LIN {X 0,Y 165.279,Z 285.697,A -85,B 0,C 180,E1 -23392.213,E2 -23392.213} C_VEL
LIN {X 0,Y 165.239,Z 285.426,A -85,B 0,C 180,E1 -23392.672,E2 -23392.672} C_VEL
LIN {X 0,Y 165.636,Z 284.894,A -85,B 0,C 180,E1 -23400.003,E2 -23400.003} C_VEL
LIN {X 0,Y 165.274,Z 285.304,A -85,B 0,C 180,E1 -23407.332,E2 -23407.332} C_VEL
LIN {X 0,Y 165.239,Z 285.88,A -85,B 0,C 180,E1 -23411.981,E2 -23411.981} C_VEL
LIN {X 0,Y 165.204,Z 286.851,A -85,B 0,C 180,E1 -23417.328,E2 -23417.328} C_VEL
LIN {X 0,Y 165.354,Z 287.875,A -85,B 0,C 180,E1 -23420.922,E2 -23420.922} C_VEL
LIN {X 0,Y 166.724,Z 291.129,A -85,B 0,C 180,E1 -23423.281,E2 -23423.281} C_VEL
LIN {X 0,Y 169.93,Z 294.587,A -85,B 0,C 180,E1 -23427.064,E2 -23427.064} C_VEL
LIN {X 0,Y 171.948,Z 298.713,A -85,B 0,C 180,E1 -23429.543,E2 -23429.543} C_VEL
LIN {X 0,Y 174.222,Z 301.462,A -85,B 0,C 180,E1 -23431.708,E2 -23431.708} C_VEL
LIN {X 0,Y 176.103,Z 305.449,A -85,B 0,C 180,E1 -23433.736,E2 -23433.736} C_VEL
LIN {X 0,Y 177.62,Z 307.849,A -85,B 0,C 180,E1 -23435.139,E2 -23435.139} C_VEL
LIN {X 0,Y 180.387,Z 313.585,A -85,B 0,C 180,E1 -23437.856,E2 -23437.856} C_VEL
LIN {X 0,Y 183.198,Z 320.279,A -85,B 0,C 180,E1 -23440.708,E2 -23440.708} C_VEL
LIN {X 0,Y 185.902,Z 327.653,A -85,B 0,C 180,E1 -23443.628,E2 -23443.628} C_VEL
LIN {X 0,Y 187.357,Z 334.16,A -85,B 0,C 180,E1 -23445.893,E2 -23445.893} C_VEL
LIN {X 0,Y 187.851,Z 342.319,A -85,B 0,C 180,E1 -23448.442,E2 -23448.442} C_VEL
LIN {X 0,Y 187.472,Z 350.553,A -85,B 0,C 180,E1 -23451.036,E2 -23451.036} C_VEL
LIN {X 0,Y 186.501,Z 358.181,A -85,B 0,C 180,E1 -23453.594,E2 -23453.594} C_VEL
LIN {X 0,Y 185.205,Z 363.138,A -85,B 0,C 180,E1 -23455.306,E2 -23455.306} C_VEL
LIN {X 0,Y 180.202,Z 371.77,A -85,B 0,C 180,E1 -23458.231,E2 -23458.231} C_VEL
LIN {X 0,Y 175.803,Z 378.681,A -85,B 0,C 180,E1 -23461.334,E2 -23461.334} C_VEL
LIN {X 0,Y 172.088,Z 384.243,A -85,B 0,C 180,E1 -23464.608,E2 -23464.608} C_VEL
LIN {X 0,Y 168.804,Z 388.644,A -85,B 0,C 180,E1 -23467.994,E2 -23467.994} C_VEL
LIN {X 0,Y 166.897,Z 390.981,A -85,B 0,C 180,E1 -23470.314,E2 -23470.314} C_VEL
LIN {X 0,Y 165.302,Z 392.899,A -85,B 0,C 180,E1 -23472.686,E2 -23472.686} C_VEL
LIN {X 0,Y 164.118,Z 394.399,A -85,B 0,C 180,E1 -23475.112,E2 -23475.112} C_VEL
LIN {X 0,Y 162.46,Z 396.157,A -85,B 0,C 180,E1 -23480.036,E2 -23480.036} C_VEL
LIN {X 0,Y 161.856,Z 396.404,A -85,B 0,C 180,E1 -23485.018,E2 -23485.018} C_VEL
LIN {X 0,Y 161.843,Z 395.911,A -85,B 0,C 180,E1 -23487.511,E2 -23487.511} C_VEL
LIN {X 0,Y 161.942,Z 395.021,A -85,B 0,C 180,E1 -23490,E2 -23490} C_VEL
LIN {X 0,Y 161.84,Z 393.556,A -85,B 0,C 180,E1 -23492.769,E2 -23492.769} C_VEL
LIN {X 0,Y 161.976,Z 390.939,A -85,B 0,C 180,E1 -23496.227,E2 -23496.227} C_VEL
LIN {X 0,Y 162.403,Z 387.105,A -85,B 0,C 180,E1 -23499.968,E2 -23499.968} C_VEL
LIN {X 0,Y 163.312,Z 382.12,A -85,B 0,C 180,E1 -23503.691,E2 -23503.691} C_VEL
LIN {X 0,Y 164.882,Z 375.841,A -85,B 0,C 180,E1 -23507.359,E2 -23507.359} C_VEL
LIN {X 0,Y 167.078,Z 367.691,A -85,B 0,C 180,E1 -23511.067,E2 -23511.067} C_VEL
LIN {X 0,Y 168.85,Z 360.58,A -85,B 0,C 180,E1 -23513.689,E2 -23513.689} C_VEL
LIN {X 0,Y 171.428,Z 351.112,A -85,B 0,C 180,E1 -23516.477,E2 -23516.477} C_VEL
LIN {X 0,Y 172.232,Z 346.562,A -85,B 0,C 180,E1 -23517.655,E2 -23517.655} C_VEL
LIN {X 0,Y 172.3,Z 345.493,A -85,B 0,C 180,E1 -23517.932,E2 -23517.932} C_VEL
LIN {X 0,Y 171.915,Z 340.91,A -85,B 0,C 180,E1 -23519.161,E2 -23519.161} C_VEL
LIN {X 0,Y 170.545,Z 336.486,A -85,B 0,C 180,E1 -23520.408,E2 -23520.408} C_VEL
LIN {X 0,Y 166.885,Z 327.585,A -85,B 0,C 180,E1 -23522.844,E2 -23522.844} C_VEL
LIN {X 0,Y 165.579,Z 322.739,A -85,B 0,C 180,E1 -23523.969,E2 -23523.969} C_VEL
LIN {X 0,Y 165.325,Z 321.027,A -85,B 0,C 180,E1 -23524.313,E2 -23524.313} C_VEL
LIN {X 0,Y 163.739,Z 309.046,A -85,B 0,C 180,E1 -23526.448,E2 -23526.448} C_VEL
LIN {X 0,Y 161.215,Z 297.421,A -85,B 0,C 180,E1 -23528.304,E2 -23528.304} C_VEL
LIN {X 0,Y 159.652,Z 293.515,A -85,B 0,C 180,E1 -23528.995,E2 -23528.995} C_VEL
LIN {X 0,Y 158.483,Z 290.377,A -85,B 0,C 180,E1 -23529.519,E2 -23529.519} C_VEL
LIN {X 0,Y 158.438,Z 289.902,A -85,B 0,C 180,E1 -23529.716,E2 -23529.716} C_VEL
LIN {X 0,Y 157.715,Z 286.321,A -85,B 0,C 180,E1 -23535.477,E2 -23535.477} C_VEL
LIN {X 0,Y 157.262,Z 283.904,A -85,B 0,C 180,E1 -23539.885,E2 -23539.885} C_VEL
LIN {X 0,Y 157.276,Z 283.897,A -85,B 0,C 180,E1 -23544.482,E2 -23544.482} C_VEL
LIN {X 0,Y 157.284,Z 283.893,A -85,B 0,C 180,E1 -23548.1,E2 -23548.1} C_VEL
LIN {X 0,Y 157.31,Z 283.89,A -85,B 0,C 180,E1 -23553.461,E2 -23553.461} C_VEL
LIN {X 0,Y 157.392,Z 283.881,A -85,B 0,C 180,E1 -23559.667,E2 -23559.667} C_VEL
LIN {X 0,Y 157.44,Z 283.875,A -85,B 0,C 180,E1 -23564.461,E2 -23564.461} C_VEL
LIN {X 0,Y 157.688,Z 283.837,A -85,B 0,C 180,E1 -23569.728,E2 -23569.728} C_VEL
LIN {X 0,Y 157.765,Z 283.836,A -85,B 0,C 180,E1 -23572.317,E2 -23572.317} C_VEL
LIN {X 0,Y 158.255,Z 283.735,A -85,B 0,C 180,E1 -23579.997,E2 -23579.997} C_VEL
LIN {X 0,Y 157.806,Z 283.826,A -85,B 0,C 180,E1 -23587.675,E2 -23587.675} C_VEL
LIN {X 0,Y 157.668,Z 283.84,A -85,B 0,C 180,E1 -23591.298,E2 -23591.298} C_VEL
LIN {X 0,Y 157.448,Z 283.866,A -85,B 0,C 180,E1 -23595.531,E2 -23595.531} C_VEL
LIN {X 0,Y 157.364,Z 283.883,A -85,B 0,C 180,E1 -23600.93,E2 -23600.93} C_VEL
LIN {X 0,Y 157.305,Z 283.888,A -85,B 0,C 180,E1 -23606.679,E2 -23606.679} C_VEL
LIN {X 0,Y 157.271,Z 283.89,A -85,B 0,C 180,E1 -23612.424,E2 -23612.424} C_VEL
LIN {X 0,Y 157.318,Z 283.878,A -85,B 0,C 180,E1 -23616.475,E2 -23616.475} C_VEL
LIN {X 0,Y 157.264,Z 283.887,A -85,B 0,C 180,E1 -23622.089,E2 -23622.089} C_VEL
LIN {X 0,Y 157.223,Z 283.892,A -85,B 0,C 180,E1 -23627.894,E2 -23627.894} C_VEL
LIN {X 0,Y 157.272,Z 283.891,A -85,B 0,C 180,E1 -23633.543,E2 -23633.543} C_VEL
LIN {X 0,Y 157.276,Z 283.894,A -85,B 0,C 180,E1 -23638.1,E2 -23638.1} C_VEL
LIN {X 0,Y 157.298,Z 283.954,A -85,B 0,C 180,E1 -23643.32,E2 -23643.32} C_VEL
LIN {X 0,Y 158.336,Z 286.745,A -85,B 0,C 180,E1 -23643.813,E2 -23643.813} C_VEL
LIN {X 0,Y 159.794,Z 289.096,A -85,B 0,C 180,E1 -23644.361,E2 -23644.361} C_VEL
LIN {X 0,Y 161.784,Z 294.226,A -85,B 0,C 180,E1 -23645.342,E2 -23645.342} C_VEL
LIN {X 0,Y 164.927,Z 305.378,A -85,B 0,C 180,E1 -23647.449,E2 -23647.449} C_VEL
LIN {X 0,Y 166.797,Z 315.823,A -85,B 0,C 180,E1 -23649.548,E2 -23649.548} C_VEL
LIN {X 0,Y 167.906,Z 326.811,A -85,B 0,C 180,E1 -23652.02,E2 -23652.02} C_VEL
LIN {X 0,Y 167.891,Z 333.244,A -85,B 0,C 180,E1 -23653.587,E2 -23653.587} C_VEL
LIN {X 0,Y 165.068,Z 343.638,A -85,B 0,C 180,E1 -23656.144,E2 -23656.144} C_VEL
LIN {X 0,Y 162.84,Z 352.088,A -85,B 0,C 180,E1 -23658.801,E2 -23658.801} C_VEL
LIN {X 0,Y 160.566,Z 359.905,A -85,B 0,C 180,E1 -23661.822,E2 -23661.822} C_VEL
LIN {X 0,Y 158.265,Z 367.551,A -85,B 0,C 180,E1 -23665.543,E2 -23665.543} C_VEL
LIN {X 0,Y 156.935,Z 372.774,A -85,B 0,C 180,E1 -23668.717,E2 -23668.717} C_VEL
LIN {X 0,Y 155.776,Z 377.838,A -85,B 0,C 180,E1 -23672.586,E2 -23672.586} C_VEL
LIN {X 0,Y 154.956,Z 381.781,A -85,B 0,C 180,E1 -23676.51,E2 -23676.51} C_VEL
LIN {X 0,Y 154.432,Z 384.696,A -85,B 0,C 180,E1 -23680.488,E2 -23680.488} C_VEL
LIN {X 0,Y 154.39,Z 386.074,A -85,B 0,C 180,E1 -23683.156,E2 -23683.156} C_VEL
LIN {X 0,Y 154.746,Z 387.44,A -85,B 0,C 180,E1 -23687.507,E2 -23687.507} C_VEL
LIN {X 0,Y 155.396,Z 387.75,A -85,B 0,C 180,E1 -23691.211,E2 -23691.211} C_VEL
LIN {X 0,Y 156.252,Z 387.467,A -85,B 0,C 180,E1 -23693.878,E2 -23693.878} C_VEL
LIN {X 0,Y 157.494,Z 386.688,A -85,B 0,C 180,E1 -23696.822,E2 -23696.822} C_VEL
LIN {X 0,Y 160.357,Z 384.065,A -85,B 0,C 180,E1 -23701.73,E2 -23701.73} C_VEL
LIN {X 0,Y 162.836,Z 381.433,A -85,B 0,C 180,E1 -23704.917,E2 -23704.917} C_VEL
LIN {X 0,Y 167.024,Z 376.456,A -85,B 0,C 180,E1 -23709.135,E2 -23709.135} C_VEL
LIN {X 0,Y 171.629,Z 370.382,A -85,B 0,C 180,E1 -23712.834,E2 -23712.834} C_VEL
LIN {X 0,Y 176.146,Z 363.694,A -85,B 0,C 180,E1 -23715.903,E2 -23715.903} C_VEL
LIN {X 0,Y 181.013,Z 355.688,A -85,B 0,C 180,E1 -23718.701,E2 -23718.701} C_VEL
LIN {X 0,Y 182.586,Z 352.612,A -85,B 0,C 180,E1 -23719.661,E2 -23719.661} C_VEL
LIN {X 0,Y 183.295,Z 344.321,A -85,B 0,C 180,E1 -23722.89,E2 -23722.89} C_VEL
LIN {X 0,Y 183.118,Z 337.344,A -85,B 0,C 180,E1 -23725.525,E2 -23725.525} C_VEL
LIN {X 0,Y 182.209,Z 330.915,A -85,B 0,C 180,E1 -23728.053,E2 -23728.053} C_VEL
LIN {X 0,Y 180.3,Z 324.284,A -85,B 0,C 180,E1 -23730.936,E2 -23730.936} C_VEL
LIN {X 0,Y 177.754,Z 317.303,A -85,B 0,C 180,E1 -23734.223,E2 -23734.223} C_VEL
LIN {X 0,Y 175.156,Z 311.906,A -85,B 0,C 180,E1 -23737.163,E2 -23737.163} C_VEL
LIN {X 0,Y 172.885,Z 307.483,A -85,B 0,C 180,E1 -23739.789,E2 -23739.789} C_VEL
LIN {X 0,Y 170,Z 302.603,A -85,B 0,C 180,E1 -23743.182,E2 -23743.182} C_VEL
LIN {X 0,Y 167.954,Z 299.607,A -85,B 0,C 180,E1 -23745.694,E2 -23745.694} C_VEL
LIN {X 0,Y 167.153,Z 297.848,A -85,B 0,C 180,E1 -23746.942,E2 -23746.942} C_VEL
LIN {X 0,Y 164.506,Z 294.958,A -85,B 0,C 180,E1 -23750.629,E2 -23750.629} C_VEL
LIN {X 0,Y 163.297,Z 292.219,A -85,B 0,C 180,E1 -23753.206,E2 -23753.206} C_VEL
LIN {X 0,Y 160.482,Z 289.774,A -85,B 0,C 180,E1 -23760.003,E2 -23760.003} C_VEL
LIN {X 0,Y 159.59,Z 289.477,A -85,B 0,C 180,E1 -23765.056,E2 -23765.056} C_VEL
LIN {X 0,Y 159.736,Z 289.995,A -85,B 0,C 180,E1 -23769.5,E2 -23769.5} C_VEL
LIN {X 0,Y 163.477,Z 294.396,A -85,B 0,C 180,E1 -23780.119,E2 -23780.119} C_VEL
LIN {X 0,Y 164.634,Z 297.606,A -85,B 0,C 180,E1 -23782.597,E2 -23782.597} C_VEL
LIN {X 0,Y 167.62,Z 301.396,A -85,B 0,C 180,E1 -23786.625,E2 -23786.625} C_VEL
LIN {X 0,Y 168.954,Z 304.57,A -85,B 0,C 180,E1 -23788.583,E2 -23788.583} C_VEL
LIN {X 0,Y 171.064,Z 307.424,A -85,B 0,C 180,E1 -23790.904,E2 -23790.904} C_VEL
LIN {X 0,Y 172.593,Z 311.035,A -85,B 0,C 180,E1 -23792.85,E2 -23792.85} C_VEL
LIN {X 0,Y 174.036,Z 313.646,A -85,B 0,C 180,E1 -23794.43,E2 -23794.43} C_VEL
LIN {X 0,Y 177.073,Z 320.756,A -85,B 0,C 180,E1 -23797.967,E2 -23797.967} C_VEL
LIN {X 0,Y 179.999,Z 328.949,A -85,B 0,C 180,E1 -23801.59,E2 -23801.59} C_VEL
LIN {X 0,Y 181.606,Z 335.39,A -85,B 0,C 180,E1 -23804.157,E2 -23804.157} C_VEL
LIN {X 0,Y 182.117,Z 340.664,A -85,B 0,C 180,E1 -23806.004,E2 -23806.004} C_VEL
LIN {X 0,Y 181.912,Z 348.306,A -85,B 0,C 180,E1 -23808.539,E2 -23808.539} C_VEL
LIN {X 0,Y 180.859,Z 356.997,A -85,B 0,C 180,E1 -23811.558,E2 -23811.558} C_VEL
LIN {X 0,Y 179.336,Z 363.575,A -85,B 0,C 180,E1 -23813.998,E2 -23813.998} C_VEL
LIN {X 0,Y 174.219,Z 372.049,A -85,B 0,C 180,E1 -23817.004,E2 -23817.004} C_VEL
LIN {X 0,Y 169.599,Z 378.868,A -85,B 0,C 180,E1 -23820.182,E2 -23820.182} C_VEL
LIN {X 0,Y 165.702,Z 384.352,A -85,B 0,C 180,E1 -23823.556,E2 -23823.556} C_VEL
LIN {X 0,Y 162.216,Z 388.682,A -85,B 0,C 180,E1 -23827.051,E2 -23827.051} C_VEL
LIN {X 0,Y 160.216,Z 390.985,A -85,B 0,C 180,E1 -23829.457,E2 -23829.457} C_VEL
LIN {X 0,Y 158.515,Z 392.869,A -85,B 0,C 180,E1 -23831.92,E2 -23831.92} C_VEL
LIN {X 0,Y 156.214,Z 395.344,A -85,B 0,C 180,E1 -23837.001,E2 -23837.001} C_VEL
LIN {X 0,Y 154.98,Z 396.286,A -85,B 0,C 180,E1 -23842.181,E2 -23842.181} C_VEL
LIN {X 0,Y 154.765,Z 396.165,A -85,B 0,C 180,E1 -23844.789,E2 -23844.789} C_VEL
LIN {X 0,Y 154.749,Z 395.547,A -85,B 0,C 180,E1 -23847.69,E2 -23847.69} C_VEL
LIN {X 0,Y 154.86,Z 394.714,A -85,B 0,C 180,E1 -23850,E2 -23850} C_VEL
LIN {X 0,Y 154.747,Z 393.38,A -85,B 0,C 180,E1 -23852.603,E2 -23852.603} C_VEL
LIN {X 0,Y 154.902,Z 390.534,A -85,B 0,C 180,E1 -23856.513,E2 -23856.513} C_VEL
LIN {X 0,Y 155.4,Z 386.632,A -85,B 0,C 180,E1 -23860.422,E2 -23860.422} C_VEL
LIN {X 0,Y 156.383,Z 381.571,A -85,B 0,C 180,E1 -23864.31,E2 -23864.31} C_VEL
LIN {X 0,Y 158.055,Z 375.197,A -85,B 0,C 180,E1 -23868.135,E2 -23868.135} C_VEL
LIN {X 0,Y 160.353,Z 367.189,A -85,B 0,C 180,E1 -23871.872,E2 -23871.872} C_VEL
LIN {X 0,Y 161.778,Z 361.497,A -85,B 0,C 180,E1 -23874.085,E2 -23874.085} C_VEL
LIN {X 0,Y 164.457,Z 352.241,A -85,B 0,C 180,E1 -23877.003,E2 -23877.003} C_VEL
LIN {X 0,Y 165.445,Z 347.846,A -85,B 0,C 180,E1 -23878.201,E2 -23878.201} C_VEL
LIN {X 0,Y 165.907,Z 337.311,A -85,B 0,C 180,E1 -23880.89,E2 -23880.89} C_VEL
LIN {X 0,Y 165.735,Z 326.673,A -85,B 0,C 180,E1 -23883.205,E2 -23883.205} C_VEL
LIN {X 0,Y 165.325,Z 321.027,A -85,B 0,C 180,E1 -23884.313,E2 -23884.313} C_VEL
LIN {X 0,Y 164.169,Z 316.085,A -85,B 0,C 180,E1 -23885.362,E2 -23885.362} C_VEL
LIN {X 0,Y 162.1,Z 311.515,A -85,B 0,C 180,E1 -23886.482,E2 -23886.482} C_VEL
LIN {X 0,Y 155.231,Z 299.656,A -85,B 0,C 180,E1 -23889.493,E2 -23889.493} C_VEL
LIN {X 0,Y 153.815,Z 296.375,A -85,B 0,C 180,E1 -23890.169,E2 -23890.169} C_VEL
LIN {X 0,Y 152.408,Z 293.22,A -85,B 0,C 180,E1 -23890.811,E2 -23890.811} C_VEL
LIN {X 0,Y 151.237,Z 290.151,A -85,B 0,C 180,E1 -23891.381,E2 -23891.381} C_VEL
LIN {X 0,Y 151.175,Z 289.718,A -85,B 0,C 180,E1 -23891.501,E2 -23891.501} C_VEL
LIN {X 0,Y 150.68,Z 287.319,A -85,B 0,C 180,E1 -23895.599,E2 -23895.599} C_VEL
LIN {X 0,Y 150.217,Z 284.782,A -85,B 0,C 180,E1 -23900.394,E2 -23900.394} C_VEL
LIN {X 0,Y 150.187,Z 284.777,A -85,B 0,C 180,E1 -23905.834,E2 -23905.834} C_VEL
LIN {X 0,Y 150.192,Z 284.773,A -85,B 0,C 180,E1 -23909.017,E2 -23909.017} C_VEL
LIN {X 0,Y 150.24,Z 284.772,A -85,B 0,C 180,E1 -23912.72,E2 -23912.72} C_VEL
LIN {X 0,Y 150.35,Z 284.758,A -85,B 0,C 180,E1 -23919.207,E2 -23919.207} C_VEL
LIN {X 0,Y 150.351,Z 284.754,A -85,B 0,C 180,E1 -23923.709,E2 -23923.709} C_VEL
LIN {X 0,Y 150.61,Z 284.717,A -85,B 0,C 180,E1 -23929.239,E2 -23929.239} C_VEL
LIN {X 0,Y 150.702,Z 284.715,A -85,B 0,C 180,E1 -23931.955,E2 -23931.955} C_VEL
LIN {X 0,Y 151.215,Z 284.61,A -85,B 0,C 180,E1 -23939.997,E2 -23939.997} C_VEL
LIN {X 0,Y 150.74,Z 284.704,A -85,B 0,C 180,E1 -23948.037,E2 -23948.037} C_VEL
LIN {X 0,Y 150.602,Z 284.721,A -85,B 0,C 180,E1 -23951.488,E2 -23951.488} C_VEL
LIN {X 0,Y 150.355,Z 284.747,A -85,B 0,C 180,E1 -23956.284,E2 -23956.284} C_VEL
LIN {X 0,Y 150.345,Z 284.757,A -85,B 0,C 180,E1 -23960.789,E2 -23960.789} C_VEL
LIN {X 0,Y 150.236,Z 284.77,A -85,B 0,C 180,E1 -23967.278,E2 -23967.278} C_VEL
LIN {X 0,Y 150.212,Z 284.77,A -85,B 0,C 180,E1 -23972.632,E2 -23972.632} C_VEL
LIN {X 0,Y 150.228,Z 284.763,A -85,B 0,C 180,E1 -23977.453,E2 -23977.453} C_VEL
LIN {X 0,Y 150.209,Z 284.767,A -85,B 0,C 180,E1 -23981.531,E2 -23981.531} C_VEL
LIN {X 0,Y 150.16,Z 284.779,A -85,B 0,C 180,E1 -23985.409,E2 -23985.409} C_VEL
LIN {X 0,Y 150.158,Z 284.776,A -85,B 0,C 180,E1 -23989.062,E2 -23989.062} C_VEL
LIN {X 0,Y 150.207,Z 284.769,A -85,B 0,C 180,E1 -23992.688,E2 -23992.688} C_VEL
LIN {X 0,Y 150.202,Z 284.776,A -85,B 0,C 180,E1 -23997.369,E2 -23997.369} C_VEL
LIN {X 0,Y 150.218,Z 284.931,A -85,B 0,C 180,E1 -24001.537,E2 -24001.537} C_VEL
LIN {X 0,Y 151.328,Z 287.771,A -85,B 0,C 180,E1 -24002.102,E2 -24002.102} C_VEL
LIN {X 0,Y 152.91,Z 290.388,A -85,B 0,C 180,E1 -24002.777,E2 -24002.777} C_VEL
LIN {X 0,Y 155.092,Z 294.395,A -85,B 0,C 180,E1 -24003.773,E2 -24003.773} C_VEL
LIN {X 0,Y 158.216,Z 305.436,A -85,B 0,C 180,E1 -24006.011,E2 -24006.011} C_VEL
LIN {X 0,Y 160.146,Z 315.532,A -85,B 0,C 180,E1 -24008.179,E2 -24008.179} C_VEL
LIN {X 0,Y 161.307,Z 327.158,A -85,B 0,C 180,E1 -24010.928,E2 -24010.928} C_VEL
LIN {X 0,Y 161.399,Z 333.533,A -85,B 0,C 180,E1 -24012.581,E2 -24012.581} C_VEL
LIN {X 0,Y 158.469,Z 343.908,A -85,B 0,C 180,E1 -24015.226,E2 -24015.226} C_VEL
LIN {X 0,Y 155.866,Z 353.18,A -85,B 0,C 180,E1 -24018.293,E2 -24018.293} C_VEL
LIN {X 0,Y 153.119,Z 362.192,A -85,B 0,C 180,E1 -24022.085,E2 -24022.085} C_VEL
LIN {X 0,Y 150.827,Z 369.472,A -85,B 0,C 180,E1 -24025.992,E2 -24025.992} C_VEL
LIN {X 0,Y 149.296,Z 375.275,A -85,B 0,C 180,E1 -24030,E2 -24030} C_VEL
LIN {X 0,Y 148.244,Z 380.142,A -85,B 0,C 180,E1 -24034.395,E2 -24034.395} C_VEL
LIN {X 0,Y 147.562,Z 383.35,A -85,B 0,C 180,E1 -24038.214,E2 -24038.214} C_VEL
LIN {X 0,Y 147.307,Z 385.097,A -85,B 0,C 180,E1 -24041.001,E2 -24041.001} C_VEL
LIN {X 0,Y 147.305,Z 386.432,A -85,B 0,C 180,E1 -24043.801,E2 -24043.801} C_VEL
LIN {X 0,Y 147.7,Z 387.627,A -85,B 0,C 180,E1 -24047.9,E2 -24047.9} C_VEL
LIN {X 0,Y 148.572,Z 387.934,A -85,B 0,C 180,E1 -24052.236,E2 -24052.236} C_VEL
LIN {X 0,Y 150.68,Z 386.928,A -85,B 0,C 180,E1 -24057.609,E2 -24057.609} C_VEL
LIN {X 0,Y 152.306,Z 385.66,A -85,B 0,C 180,E1 -24060.502,E2 -24060.502} C_VEL
LIN {X 0,Y 155.126,Z 383.039,A -85,B 0,C 180,E1 -24064.493,E2 -24064.493} C_VEL
LIN {X 0,Y 158.644,Z 379.339,A -85,B 0,C 180,E1 -24068.33,E2 -24068.33} C_VEL
LIN {X 0,Y 162.816,Z 374.444,A -85,B 0,C 180,E1 -24071.993,E2 -24071.993} C_VEL
LIN {X 0,Y 167.586,Z 368.203,A -85,B 0,C 180,E1 -24075.472,E2 -24075.472} C_VEL
LIN {X 0,Y 172.948,Z 360.372,A -85,B 0,C 180,E1 -24078.743,E2 -24078.743} C_VEL
LIN {X 0,Y 175.983,Z 355.415,A -85,B 0,C 180,E1 -24080.385,E2 -24080.385} C_VEL
LIN {X 0,Y 176.65,Z 353.79,A -85,B 0,C 180,E1 -24080.972,E2 -24080.972} C_VEL
LIN {X 0,Y 177.466,Z 345.906,A -85,B 0,C 180,E1 -24084.263,E2 -24084.263} C_VEL
LIN {X 0,Y 177.398,Z 339.024,A -85,B 0,C 180,E1 -24087.079,E2 -24087.079} C_VEL
LIN {X 0,Y 176.603,Z 333.443,A -85,B 0,C 180,E1 -24089.513,E2 -24089.513} C_VEL
LIN {X 0,Y 174.57,Z 326.081,A -85,B 0,C 180,E1 -24093.072,E2 -24093.072} C_VEL
LIN {X 0,Y 173.443,Z 322.671,A -85,B 0,C 180,E1 -24094.823,E2 -24094.823} C_VEL
LIN {X 0,Y 170.081,Z 314.794,A -85,B 0,C 180,E1 -24099.44,E2 -24099.44} C_VEL
LIN {X 0,Y 167.532,Z 309.812,A -85,B 0,C 180,E1 -24102.927,E2 -24102.927} C_VEL
LIN {X 0,Y 165.073,Z 305.679,A -85,B 0,C 180,E1 -24106.461,E2 -24106.461} C_VEL
LIN {X 0,Y 164.4,Z 304.169,A -85,B 0,C 180,E1 -24107.661,E2 -24107.661} C_VEL
LIN {X 0,Y 162.18,Z 301.405,A -85,B 0,C 180,E1 -24111.279,E2 -24111.279} C_VEL
LIN {X 0,Y 161.339,Z 299.019,A -85,B 0,C 180,E1 -24113.515,E2 -24113.515} C_VEL
LIN {X 0,Y 158.914,Z 296.764,A -85,B 0,C 180,E1 -24120.003,E2 -24120.003} C_VEL
LIN {X 0,Y 158.076,Z 296.407,A -85,B 0,C 180,E1 -24125.104,E2 -24125.104} C_VEL
LIN {X 0,Y 158.217,Z 296.981,A -85,B 0,C 180,E1 -24129.592,E2 -24129.592} C_VEL
LIN {X 0,Y 161.336,Z 301.158,A -85,B 0,C 180,E1 -24139.568,E2 -24139.568} C_VEL
LIN {X 0,Y 162.59,Z 304.634,A -85,B 0,C 180,E1 -24142.561,E2 -24142.561} C_VEL
LIN {X 0,Y 164.393,Z 307.016,A -85,B 0,C 180,E1 -24145.313,E2 -24145.313} C_VEL
LIN {X 0,Y 166.477,Z 311.553,A -85,B 0,C 180,E1 -24148.62,E2 -24148.62} C_VEL
LIN {X 0,Y 167.728,Z 313.396,A -85,B 0,C 180,E1 -24150.189,E2 -24150.189} C_VEL
LIN {X 0,Y 169.431,Z 317.477,A -85,B 0,C 180,E1 -24152.635,E2 -24152.635} C_VEL
LIN {X 0,Y 172.097,Z 324.058,A -85,B 0,C 180,E1 -24156.312,E2 -24156.312} C_VEL
LIN {X 0,Y 174.688,Z 331.962,A -85,B 0,C 180,E1 -24160.148,E2 -24160.148} C_VEL
LIN {X 0,Y 176.065,Z 337.901,A -85,B 0,C 180,E1 -24162.737,E2 -24162.737} C_VEL
LIN {X 0,Y 176.53,Z 343.79,A -85,B 0,C 180,E1 -24165.02,E2 -24165.02} C_VEL
LIN {X 0,Y 176.14,Z 350.118,A -85,B 0,C 180,E1 -24167.291,E2 -24167.291} C_VEL
LIN {X 0,Y 175.028,Z 357.533,A -85,B 0,C 180,E1 -24170.026,E2 -24170.026} C_VEL
LIN {X 0,Y 173.491,Z 364.027,A -85,B 0,C 180,E1 -24172.582,E2 -24172.582} C_VEL
LIN {X 0,Y 171.915,Z 366.973,A -85,B 0,C 180,E1 -24173.647,E2 -24173.647} C_VEL
LIN {X 0,Y 166.627,Z 374.767,A -85,B 0,C 180,E1 -24176.75,E2 -24176.75} C_VEL
LIN {X 0,Y 162.025,Z 381,A -85,B 0,C 180,E1 -24180.066,E2 -24180.066} C_VEL
LIN {X 0,Y 158.062,Z 386.018,A -85,B 0,C 180,E1 -24183.601,E2 -24183.601} C_VEL
LIN {X 0,Y 154.617,Z 389.92,A -85,B 0,C 180,E1 -24187.272,E2 -24187.272} C_VEL
LIN {X 0,Y 151.764,Z 392.823,A -85,B 0,C 180,E1 -24191.086,E2 -24191.086} C_VEL
LIN {X 0,Y 149.267,Z 395.22,A -85,B 0,C 180,E1 -24196.384,E2 -24196.384} C_VEL
LIN {X 0,Y 147.949,Z 396.094,A -85,B 0,C 180,E1 -24201.807,E2 -24201.807} C_VEL
LIN {X 0,Y 147.696,Z 395.919,A -85,B 0,C 180,E1 -24204.539,E2 -24204.539} C_VEL
LIN {X 0,Y 147.683,Z 395.145,A -85,B 0,C 180,E1 -24208.022,E2 -24208.022} C_VEL
LIN {X 0,Y 147.772,Z 394.406,A -85,B 0,C 180,E1 -24210,E2 -24210} C_VEL
LIN {X 0,Y 147.652,Z 393.038,A -85,B 0,C 180,E1 -24212.728,E2 -24212.728} C_VEL
LIN {X 0,Y 147.82,Z 390.127,A -85,B 0,C 180,E1 -24216.826,E2 -24216.826} C_VEL
LIN {X 0,Y 148.378,Z 386.154,A -85,B 0,C 180,E1 -24220.921,E2 -24220.921} C_VEL
LIN {X 0,Y 149.676,Z 380.006,A -85,B 0,C 180,E1 -24225.663,E2 -24225.663} C_VEL
LIN {X 0,Y 151.661,Z 373.28,A -85,B 0,C 180,E1 -24229.631,E2 -24229.631} C_VEL
LIN {X 0,Y 154.074,Z 364.891,A -85,B 0,C 180,E1 -24233.523,E2 -24233.523} C_VEL
LIN {X 0,Y 156.332,Z 357.377,A -85,B 0,C 180,E1 -24236.284,E2 -24236.284} C_VEL
LIN {X 0,Y 158.657,Z 349.035,A -85,B 0,C 180,E1 -24238.798,E2 -24238.798} C_VEL
LIN {X 0,Y 159.277,Z 338.842,A -85,B 0,C 180,E1 -24241.599,E2 -24241.599} C_VEL
LIN {X 0,Y 159.274,Z 328.473,A -85,B 0,C 180,E1 -24244.027,E2 -24244.027} C_VEL
LIN {X 0,Y 158.568,Z 318.534,A -85,B 0,C 180,E1 -24246.079,E2 -24246.079} C_VEL
LIN {X 0,Y 156.654,Z 305.883,A -85,B 0,C 180,E1 -24248.397,E2 -24248.397} C_VEL
LIN {X 0,Y 155,Z 299.259,A -85,B 0,C 180,E1 -24249.569,E2 -24249.569} C_VEL
LIN {X 0,Y 153.815,Z 296.375,A -85,B 0,C 180,E1 -24250.169,E2 -24250.169} C_VEL
LIN {X 0,Y 151.997,Z 293.444,A -85,B 0,C 180,E1 -24250.956,E2 -24250.956} C_VEL
LIN {X 0,Y 148.739,Z 290.886,A -85,B 0,C 180,E1 -24252.326,E2 -24252.326} C_VEL
LIN {X 0,Y 145.603,Z 289.325,A -85,B 0,C 180,E1 -24254.025,E2 -24254.025} C_VEL
LIN {X 0,Y 143.813,Z 288.305,A -85,B 0,C 180,E1 -24255.771,E2 -24255.771} C_VEL
LIN {X 0,Y 143.554,Z 287.878,A -85,B 0,C 180,E1 -24256.575,E2 -24256.575} C_VEL
LIN {X 0,Y 143.136,Z 285.662,A -85,B 0,C 180,E1 -24261.18,E2 -24261.18} C_VEL
LIN {X 0,Y 143.177,Z 285.65,A -85,B 0,C 180,E1 -24267.316,E2 -24267.316} C_VEL
LIN {X 0,Y 143.184,Z 285.647,A -85,B 0,C 180,E1 -24272.066,E2 -24272.066} C_VEL
LIN {X 0,Y 143.275,Z 285.64,A -85,B 0,C 180,E1 -24278.745,E2 -24278.745} C_VEL
LIN {X 0,Y 143.294,Z 285.63,A -85,B 0,C 180,E1 -24282.883,E2 -24282.883} C_VEL
LIN {X 0,Y 143.536,Z 285.598,A -85,B 0,C 180,E1 -24288.702,E2 -24288.702} C_VEL
LIN {X 0,Y 143.624,Z 285.596,A -85,B 0,C 180,E1 -24291.555,E2 -24291.555} C_VEL
LIN {X 0,Y 144.174,Z 285.486,A -85,B 0,C 180,E1 -24299.997,E2 -24299.997} C_VEL
LIN {X 0,Y 143.659,Z 285.585,A -85,B 0,C 180,E1 -24308.436,E2 -24308.436} C_VEL
LIN {X 0,Y 143.544,Z 285.601,A -85,B 0,C 180,E1 -24311.709,E2 -24311.709} C_VEL
LIN {X 0,Y 143.295,Z 285.625,A -85,B 0,C 180,E1 -24317.11,E2 -24317.11} C_VEL
LIN {X 0,Y 143.271,Z 285.637,A -85,B 0,C 180,E1 -24321.251,E2 -24321.251} C_VEL
LIN {X 0,Y 143.183,Z 285.646,A -85,B 0,C 180,E1 -24327.933,E2 -24327.933} C_VEL
LIN {X 0,Y 143.163,Z 285.65,A -85,B 0,C 180,E1 -24333.433,E2 -24333.433} C_VEL
LIN {X 0,Y 143.113,Z 285.656,A -85,B 0,C 180,E1 -24339.668,E2 -24339.668} C_VEL
LIN {X 0,Y 143.111,Z 285.651,A -85,B 0,C 180,E1 -24343.429,E2 -24343.429} C_VEL
LIN {X 0,Y 143.077,Z 285.654,A -85,B 0,C 180,E1 -24347.454,E2 -24347.454} C_VEL
LIN {X 0,Y 143.101,Z 285.656,A -85,B 0,C 180,E1 -24351.788,E2 -24351.788} C_VEL
LIN {X 0,Y 143.17,Z 285.652,A -85,B 0,C 180,E1 -24357.319,E2 -24357.319} C_VEL
LIN {X 0,Y 143.146,Z 285.655,A -85,B 0,C 180,E1 -24359.484,E2 -24359.484} C_VEL
LIN {X 0,Y 144.206,Z 288.601,A -85,B 0,C 180,E1 -24360.132,E2 -24360.132} C_VEL
LIN {X 0,Y 145.517,Z 290.518,A -85,B 0,C 180,E1 -24360.727,E2 -24360.727} C_VEL
LIN {X 0,Y 149.602,Z 298.302,A -85,B 0,C 180,E1 -24362.854,E2 -24362.854} C_VEL
LIN {X 0,Y 152.227,Z 308.298,A -85,B 0,C 180,E1 -24365.085,E2 -24365.085} C_VEL
LIN {X 0,Y 153.769,Z 316.876,A -85,B 0,C 180,E1 -24367.076,E2 -24367.076} C_VEL
LIN {X 0,Y 154.768,Z 327.484,A -85,B 0,C 180,E1 -24369.742,E2 -24369.742} C_VEL
LIN {X 0,Y 154.885,Z 333.83,A -85,B 0,C 180,E1 -24371.481,E2 -24371.481} C_VEL
LIN {X 0,Y 152.213,Z 343.103,A -85,B 0,C 180,E1 -24373.917,E2 -24373.917} C_VEL
LIN {X 0,Y 149.458,Z 352.596,A -85,B 0,C 180,E1 -24377.094,E2 -24377.094} C_VEL
LIN {X 0,Y 146.498,Z 361.755,A -85,B 0,C 180,E1 -24381.03,E2 -24381.03} C_VEL
LIN {X 0,Y 144.035,Z 369.147,A -85,B 0,C 180,E1 -24385.102,E2 -24385.102} C_VEL
LIN {X 0,Y 142.663,Z 374.143,A -85,B 0,C 180,E1 -24388.588,E2 -24388.588} C_VEL
LIN {X 0,Y 141.467,Z 379.006,A -85,B 0,C 180,E1 -24392.847,E2 -24392.847} C_VEL
LIN {X 0,Y 140.61,Z 382.764,A -85,B 0,C 180,E1 -24397.178,E2 -24397.178} C_VEL
LIN {X 0,Y 140.179,Z 385.498,A -85,B 0,C 180,E1 -24401.568,E2 -24401.568} C_VEL
LIN {X 0,Y 140.251,Z 386.789,A -85,B 0,C 180,E1 -24404.51,E2 -24404.51} C_VEL
LIN {X 0,Y 140.647,Z 387.81,A -85,B 0,C 180,E1 -24408.315,E2 -24408.315} C_VEL
LIN {X 0,Y 141.768,Z 388.119,A -85,B 0,C 180,E1 -24413.365,E2 -24413.365} C_VEL
LIN {X 0,Y 143.889,Z 387.169,A -85,B 0,C 180,E1 -24418.465,E2 -24418.465} C_VEL
LIN {X 0,Y 145.956,Z 385.67,A -85,B 0,C 180,E1 -24421.982,E2 -24421.982} C_VEL
LIN {X 0,Y 147.937,Z 383.99,A -85,B 0,C 180,E1 -24424.755,E2 -24424.755} C_VEL
LIN {X 0,Y 151.551,Z 380.567,A -85,B 0,C 180,E1 -24428.758,E2 -24428.758} C_VEL
LIN {X 0,Y 155.806,Z 375.99,A -85,B 0,C 180,E1 -24432.578,E2 -24432.578} C_VEL
LIN {X 0,Y 161.498,Z 369.065,A -85,B 0,C 180,E1 -24436.703,E2 -24436.703} C_VEL
LIN {X 0,Y 167.174,Z 361.251,A -85,B 0,C 180,E1 -24440.104,E2 -24440.104} C_VEL
LIN {X 0,Y 170.265,Z 356.506,A -85,B 0,C 180,E1 -24441.75,E2 -24441.75} C_VEL
LIN {X 0,Y 171.145,Z 352.622,A -85,B 0,C 180,E1 -24443.46,E2 -24443.46} C_VEL
LIN {X 0,Y 171.838,Z 344.706,A -85,B 0,C 180,E1 -24446.971,E2 -24446.971} C_VEL
LIN {X 0,Y 171.47,Z 338.553,A -85,B 0,C 180,E1 -24449.798,E2 -24449.798} C_VEL
LIN {X 0,Y 170.16,Z 332.38,A -85,B 0,C 180,E1 -24452.982,E2 -24452.982} C_VEL
LIN {X 0,Y 168.437,Z 326.62,A -85,B 0,C 180,E1 -24456.217,E2 -24456.217} C_VEL
LIN {X 0,Y 166.103,Z 320.229,A -85,B 0,C 180,E1 -24460.218,E2 -24460.218} C_VEL
LIN {X 0,Y 163.905,Z 315.435,A -85,B 0,C 180,E1 -24463.82,E2 -24463.82} C_VEL
LIN {X 0,Y 161.183,Z 310.155,A -85,B 0,C 180,E1 -24468.688,E2 -24468.688} C_VEL
LIN {X 0,Y 158.51,Z 305.379,A -85,B 0,C 180,E1 -24474.916,E2 -24474.916} C_VEL
LIN {X 0,Y 156.964,Z 303.638,A -85,B 0,C 180,E1 -24480.003,E2 -24480.003} C_VEL
LIN {X 0,Y 156.19,Z 303.246,A -85,B 0,C 180,E1 -24485.166,E2 -24485.166} C_VEL
LIN {X 0,Y 156.328,Z 303.869,A -85,B 0,C 180,E1 -24489.708,E2 -24489.708} C_VEL
LIN {X 0,Y 158.462,Z 307.25,A -85,B 0,C 180,E1 -24498.09,E2 -24498.09} C_VEL
LIN {X 0,Y 158.937,Z 308.225,A -85,B 0,C 180,E1 -24499.371,E2 -24499.371} C_VEL
LIN {X 0,Y 160.495,Z 312.059,A -85,B 0,C 180,E1 -24503.213,E2 -24503.213} C_VEL
LIN {X 0,Y 161.249,Z 313.067,A -85,B 0,C 180,E1 -24504.463,E2 -24504.463} C_VEL
LIN {X 0,Y 164.149,Z 319.265,A -85,B 0,C 180,E1 -24509.499,E2 -24509.499} C_VEL
LIN {X 0,Y 166.356,Z 325.309,A -85,B 0,C 180,E1 -24513.316,E2 -24513.316} C_VEL
LIN {X 0,Y 168.621,Z 332.183,A -85,B 0,C 180,E1 -24517.187,E2 -24517.187} C_VEL
LIN {X 0,Y 170.163,Z 338.519,A -85,B 0,C 180,E1 -24520.361,E2 -24520.361} C_VEL
LIN {X 0,Y 170.931,Z 343.681,A -85,B 0,C 180,E1 -24522.722,E2 -24522.722} C_VEL
LIN {X 0,Y 170.729,Z 349.496,A -85,B 0,C 180,E1 -24525.035,E2 -24525.035} C_VEL
LIN {X 0,Y 169.341,Z 358.068,A -85,B 0,C 180,E1 -24528.393,E2 -24528.393} C_VEL
LIN {X 0,Y 167.696,Z 364.443,A -85,B 0,C 180,E1 -24531.051,E2 -24531.051} C_VEL
LIN {X 0,Y 167.145,Z 365.89,A -85,B 0,C 180,E1 -24531.671,E2 -24531.671} C_VEL
LIN {X 0,Y 161.617,Z 373.848,A -85,B 0,C 180,E1 -24534.819,E2 -24534.819} C_VEL
LIN {X 0,Y 157.416,Z 379.264,A -85,B 0,C 180,E1 -24537.606,E2 -24537.606} C_VEL
LIN {X 0,Y 153.108,Z 384.586,A -85,B 0,C 180,E1 -24541.187,E2 -24541.187} C_VEL
LIN {X 0,Y 149.191,Z 388.767,A -85,B 0,C 180,E1 -24544.916,E2 -24544.916} C_VEL
LIN {X 0,Y 146.992,Z 390.999,A -85,B 0,C 180,E1 -24547.512,E2 -24547.512} C_VEL
LIN {X 0,Y 145.054,Z 392.766,A -85,B 0,C 180,E1 -24550.175,E2 -24550.175} C_VEL
LIN {X 0,Y 142.343,Z 395.097,A -85,B 0,C 180,E1 -24555.708,E2 -24555.708} C_VEL
LIN {X 0,Y 141.461,Z 395.694,A -85,B 0,C 180,E1 -24558.538,E2 -24558.538} C_VEL
LIN {X 0,Y 140.913,Z 395.885,A -85,B 0,C 180,E1 -24561.395,E2 -24561.395} C_VEL
LIN {X 0,Y 140.627,Z 395.672,A -85,B 0,C 180,E1 -24564.264,E2 -24564.264} C_VEL
LIN {X 0,Y 140.611,Z 394.644,A -85,B 0,C 180,E1 -24568.57,E2 -24568.57} C_VEL
LIN {X 0,Y 140.603,Z 393.496,A -85,B 0,C 180,E1 -24571.289,E2 -24571.289} C_VEL
LIN {X 0,Y 140.765,Z 389.712,A -85,B 0,C 180,E1 -24577.17,E2 -24577.17} C_VEL
LIN {X 0,Y 141.381,Z 385.669,A -85,B 0,C 180,E1 -24581.469,E2 -24581.469} C_VEL
LIN {X 0,Y 142.809,Z 379.414,A -85,B 0,C 180,E1 -24586.437,E2 -24586.437} C_VEL
LIN {X 0,Y 144.959,Z 372.602,A -85,B 0,C 180,E1 -24590.579,E2 -24590.579} C_VEL
LIN {X 0,Y 147.09,Z 365.623,A -85,B 0,C 180,E1 -24593.962,E2 -24593.962} C_VEL
LIN {X 0,Y 149.013,Z 359.367,A -85,B 0,C 180,E1 -24596.467,E2 -24596.467} C_VEL
LIN {X 0,Y 151.801,Z 350.171,A -85,B 0,C 180,E1 -24599.466,E2 -24599.466} C_VEL
LIN {X 0,Y 152.64,Z 340.276,A -85,B 0,C 180,E1 -24602.36,E2 -24602.36} C_VEL
LIN {X 0,Y 152.792,Z 329.388,A -85,B 0,C 180,E1 -24605.095,E2 -24605.095} C_VEL
LIN {X 0,Y 152.079,Z 318.213,A -85,B 0,C 180,E1 -24607.546,E2 -24607.546} C_VEL
LIN {X 0,Y 150.561,Z 307.728,A -85,B 0,C 180,E1 -24609.624,E2 -24609.624} C_VEL
LIN {X 0,Y 149.124,Z 301.751,A -85,B 0,C 180,E1 -24610.795,E2 -24610.795} C_VEL
LIN {X 0,Y 145.624,Z 293.713,A -85,B 0,C 180,E1 -24612.644,E2 -24612.644} C_VEL
LIN {X 0,Y 144.161,Z 290.708,A -85,B 0,C 180,E1 -24613.365,E2 -24613.365} C_VEL
LIN {X 0,Y 143.888,Z 289.469,A -85,B 0,C 180,E1 -24613.639,E2 -24613.639} C_VEL
LIN {X 0,Y 143.554,Z 287.878,A -85,B 0,C 180,E1 -24616.575,E2 -24616.575} C_VEL
LIN {X 0,Y 142.743,Z 286.937,A -85,B 0,C 180,E1 -24618.874,E2 -24618.874} C_VEL
LIN {X 0,Y 141.066,Z 286.484,A -85,B 0,C 180,E1 -24621.163,E2 -24621.163} C_VEL
LIN {X 0,Y 136.393,Z 286.504,A -85,B 0,C 180,E1 -24627.517,E2 -24627.517} C_VEL
LIN {X 0,Y 136.047,Z 286.533,A -85,B 0,C 180,E1 -24629.202,E2 -24629.202} C_VEL
LIN {X 0,Y 136.14,Z 286.525,A -85,B 0,C 180,E1 -24632.311,E2 -24632.311} C_VEL
LIN {X 0,Y 136.242,Z 286.516,A -85,B 0,C 180,E1 -24638.829,E2 -24638.829} C_VEL
LIN {X 0,Y 136.262,Z 286.514,A -85,B 0,C 180,E1 -24645.052,E2 -24645.052} C_VEL
LIN {X 0,Y 136.43,Z 286.484,A -85,B 0,C 180,E1 -24648.164,E2 -24648.164} C_VEL
LIN {X 0,Y 136.55,Z 286.477,A -85,B 0,C 180,E1 -24651.114,E2 -24651.114} C_VEL
LIN {X 0,Y 137.13,Z 286.362,A -85,B 0,C 180,E1 -24659.996,E2 -24659.996} C_VEL
LIN {X 0,Y 136.587,Z 286.464,A -85,B 0,C 180,E1 -24668.876,E2 -24668.876} C_VEL
LIN {X 0,Y 136.487,Z 286.481,A -85,B 0,C 180,E1 -24671.951,E2 -24671.951} C_VEL
LIN {X 0,Y 136.236,Z 286.507,A -85,B 0,C 180,E1 -24678.027,E2 -24678.027} C_VEL
LIN {X 0,Y 136.192,Z 286.516,A -85,B 0,C 180,E1 -24681.745,E2 -24681.745} C_VEL
LIN {X 0,Y 136.093,Z 286.527,A -85,B 0,C 180,E1 -24688.612,E2 -24688.612} C_VEL
LIN {X 0,Y 136.076,Z 286.53,A -85,B 0,C 180,E1 -24694.615,E2 -24694.615} C_VEL
LIN {X 0,Y 136.081,Z 286.533,A -85,B 0,C 180,E1 -24699.225,E2 -24699.225} C_VEL
LIN {X 0,Y 136.045,Z 286.532,A -85,B 0,C 180,E1 -24703.679,E2 -24703.679} C_VEL
LIN {X 0,Y 136.038,Z 286.53,A -85,B 0,C 180,E1 -24707.81,E2 -24707.81} C_VEL
LIN {X 0,Y 136.05,Z 286.534,A -85,B 0,C 180,E1 -24711.693,E2 -24711.693} C_VEL
LIN {X 0,Y 136.135,Z 286.528,A -85,B 0,C 180,E1 -24717.228,E2 -24717.228} C_VEL
LIN {X 0,Y 137.141,Z 289.445,A -85,B 0,C 180,E1 -24717.926,E2 -24717.926} C_VEL
LIN {X 0,Y 138.625,Z 291.641,A -85,B 0,C 180,E1 -24718.699,E2 -24718.699} C_VEL
LIN {X 0,Y 143.769,Z 301.122,A -85,B 0,C 180,E1 -24721.624,E2 -24721.624} C_VEL
LIN {X 0,Y 146.049,Z 309.869,A -85,B 0,C 180,E1 -24723.79,E2 -24723.79} C_VEL
LIN {X 0,Y 147.572,Z 319.585,A -85,B 0,C 180,E1 -24726.23,E2 -24726.23} C_VEL
LIN {X 0,Y 148.329,Z 330.446,A -85,B 0,C 180,E1 -24729.185,E2 -24729.185} C_VEL
LIN {X 0,Y 148.27,Z 335.351,A -85,B 0,C 180,E1 -24730.622,E2 -24730.622} C_VEL
LIN {X 0,Y 145.413,Z 344.414,A -85,B 0,C 180,E1 -24733.143,E2 -24733.143} C_VEL
LIN {X 0,Y 142.531,Z 353.662,A -85,B 0,C 180,E1 -24736.455,E2 -24736.455} C_VEL
LIN {X 0,Y 139.946,Z 361.302,A -85,B 0,C 180,E1 -24739.877,E2 -24739.877} C_VEL
LIN {X 0,Y 137.285,Z 368.81,A -85,B 0,C 180,E1 -24744.123,E2 -24744.123} C_VEL
LIN {X 0,Y 135.532,Z 374.817,A -85,B 0,C 180,E1 -24748.514,E2 -24748.514} C_VEL
LIN {X 0,Y 134.317,Z 379.581,A -85,B 0,C 180,E1 -24752.999,E2 -24752.999} C_VEL
LIN {X 0,Y 133.434,Z 383.25,A -85,B 0,C 180,E1 -24757.566,E2 -24757.566} C_VEL
LIN {X 0,Y 133.065,Z 385.896,A -85,B 0,C 180,E1 -24762.196,E2 -24762.196} C_VEL
LIN {X 0,Y 133.221,Z 387.14,A -85,B 0,C 180,E1 -24765.293,E2 -24765.293} C_VEL
LIN {X 0,Y 133.594,Z 387.991,A -85,B 0,C 180,E1 -24768.763,E2 -24768.763} C_VEL
LIN {X 0,Y 135.018,Z 388.305,A -85,B 0,C 180,E1 -24774.608,E2 -24774.608} C_VEL
LIN {X 0,Y 137.148,Z 387.406,A -85,B 0,C 180,E1 -24779.416,E2 -24779.416} C_VEL
LIN {X 0,Y 139.716,Z 385.68,A -85,B 0,C 180,E1 -24783.594,E2 -24783.594} C_VEL
LIN {X 0,Y 143.761,Z 382.336,A -85,B 0,C 180,E1 -24788.545,E2 -24788.545} C_VEL
LIN {X 0,Y 148.825,Z 377.412,A -85,B 0,C 180,E1 -24793.214,E2 -24793.214} C_VEL
LIN {X 0,Y 154.774,Z 370.823,A -85,B 0,C 180,E1 -24797.549,E2 -24797.549} C_VEL
LIN {X 0,Y 160.501,Z 363.511,A -85,B 0,C 180,E1 -24801.006,E2 -24801.006} C_VEL
LIN {X 0,Y 163.976,Z 358.603,A -85,B 0,C 180,E1 -24802.839,E2 -24802.839} C_VEL
LIN {X 0,Y 164.572,Z 357.495,A -85,B 0,C 180,E1 -24803.287,E2 -24803.287} C_VEL
LIN {X 0,Y 165.843,Z 350.646,A -85,B 0,C 180,E1 -24806.575,E2 -24806.575} C_VEL
LIN {X 0,Y 166.164,Z 344.614,A -85,B 0,C 180,E1 -24809.503,E2 -24809.503} C_VEL
LIN {X 0,Y 165.633,Z 339.559,A -85,B 0,C 180,E1 -24812.181,E2 -24812.181} C_VEL
LIN {X 0,Y 164.069,Z 332.338,A -85,B 0,C 180,E1 -24816.439,E2 -24816.439} C_VEL
LIN {X 0,Y 161.93,Z 325.531,A -85,B 0,C 180,E1 -24821.007,E2 -24821.007} C_VEL
LIN {X 0,Y 160.063,Z 320.955,A -85,B 0,C 180,E1 -24824.729,E2 -24824.729} C_VEL
LIN {X 0,Y 158.343,Z 317.028,A -85,B 0,C 180,E1 -24828.482,E2 -24828.482} C_VEL
LIN {X 0,Y 156.001,Z 312.209,A -85,B 0,C 180,E1 -24834.834,E2 -24834.834} C_VEL
LIN {X 0,Y 154.603,Z 310.355,A -85,B 0,C 180,E1 -24840.003,E2 -24840.003} C_VEL
LIN {X 0,Y 154.17,Z 309.97,A -85,B 0,C 180,E1 -24842.616,E2 -24842.616} C_VEL
LIN {X 0,Y 153.933,Z 310.136,A -85,B 0,C 180,E1 -24847.876,E2 -24847.876} C_VEL
LIN {X 0,Y 155.087,Z 312.995,A -85,B 0,C 180,E1 -24855.78,E2 -24855.78} C_VEL
LIN {X 0,Y 156.008,Z 314.245,A -85,B 0,C 180,E1 -24858.385,E2 -24858.385} C_VEL
LIN {X 0,Y 157.381,Z 318.276,A -85,B 0,C 180,E1 -24862.707,E2 -24862.707} C_VEL
LIN {X 0,Y 158.439,Z 320.387,A -85,B 0,C 180,E1 -24864.926,E2 -24864.926} C_VEL
LIN {X 0,Y 160.343,Z 324.976,A -85,B 0,C 180,E1 -24868.828,E2 -24868.828} C_VEL
LIN {X 0,Y 162.452,Z 331.839,A -85,B 0,C 180,E1 -24873.379,E2 -24873.379} C_VEL
LIN {X 0,Y 163.979,Z 337.762,A -85,B 0,C 180,E1 -24876.875,E2 -24876.875} C_VEL
LIN {X 0,Y 165.2,Z 344.439,A -85,B 0,C 180,E1 -24880.451,E2 -24880.451} C_VEL
LIN {X 0,Y 165.317,Z 349.647,A -85,B 0,C 180,E1 -24882.862,E2 -24882.862} C_VEL
LIN {X 0,Y 164.123,Z 356.935,A -85,B 0,C 180,E1 -24885.906,E2 -24885.906} C_VEL
LIN {X 0,Y 161.96,Z 364.857,A -85,B 0,C 180,E1 -24889.392,E2 -24889.392} C_VEL
LIN {X 0,Y 160.725,Z 367.72,A -85,B 0,C 180,E1 -24890.653,E2 -24890.653} C_VEL
LIN {X 0,Y 154.943,Z 375.253,A -85,B 0,C 180,E1 -24893.868,E2 -24893.868} C_VEL
LIN {X 0,Y 149.686,Z 381.515,A -85,B 0,C 180,E1 -24897.481,E2 -24897.481} C_VEL
LIN {X 0,Y 145.486,Z 386.181,A -85,B 0,C 180,E1 -24901.115,E2 -24901.115} C_VEL
LIN {X 0,Y 141.596,Z 389.941,A -85,B 0,C 180,E1 -24905.047,E2 -24905.047} C_VEL
LIN {X 0,Y 138.39,Z 392.709,A -85,B 0,C 180,E1 -24909.177,E2 -24909.177} C_VEL
LIN {X 0,Y 135.449,Z 394.976,A -85,B 0,C 180,E1 -24914.964,E2 -24914.964} C_VEL
LIN {X 0,Y 134.496,Z 395.531,A -85,B 0,C 180,E1 -24917.936,E2 -24917.936} C_VEL
LIN {X 0,Y 133.555,Z 395.424,A -85,B 0,C 180,E1 -24923.959,E2 -24923.959} C_VEL
LIN {X 0,Y 133.55,Z 394.048,A -85,B 0,C 180,E1 -24929.284,E2 -24929.284} C_VEL
LIN {X 0,Y 133.475,Z 392.304,A -85,B 0,C 180,E1 -24933.018,E2 -24933.018} C_VEL
LIN {X 0,Y 133.697,Z 389.272,A -85,B 0,C 180,E1 -24937.551,E2 -24937.551} C_VEL
LIN {X 0,Y 134.379,Z 385.153,A -85,B 0,C 180,E1 -24942.075,E2 -24942.075} C_VEL
LIN {X 0,Y 135.975,Z 378.815,A -85,B 0,C 180,E1 -24947.289,E2 -24947.289} C_VEL
LIN {X 0,Y 138.289,Z 371.912,A -85,B 0,C 180,E1 -24951.62,E2 -24951.62} C_VEL
LIN {X 0,Y 140.413,Z 365.119,A -85,B 0,C 180,E1 -24955.022,E2 -24955.022} C_VEL
LIN {X 0,Y 143.326,Z 356.471,A -85,B 0,C 180,E1 -24958.48,E2 -24958.48} C_VEL
LIN {X 0,Y 145.229,Z 350.189,A -85,B 0,C 180,E1 -24960.538,E2 -24960.538} C_VEL
LIN {X 0,Y 146.111,Z 340.392,A -85,B 0,C 180,E1 -24963.56,E2 -24963.56} C_VEL
LIN {X 0,Y 146.34,Z 330.057,A -85,B 0,C 180,E1 -24966.311,E2 -24966.311} C_VEL
LIN {X 0,Y 145.79,Z 319.445,A -85,B 0,C 180,E1 -24968.805,E2 -24968.805} C_VEL
LIN {X 0,Y 144.508,Z 309.374,A -85,B 0,C 180,E1 -24970.955,E2 -24970.955} C_VEL
LIN {X 0,Y 143.415,Z 304.963,A -85,B 0,C 180,E1 -24971.936,E2 -24971.936} C_VEL
LIN {X 0,Y 140.487,Z 297.857,A -85,B 0,C 180,E1 -24973.755,E2 -24973.755} C_VEL
LIN {X 0,Y 138.233,Z 293.245,A -85,B 0,C 180,E1 -24974.997,E2 -24974.997} C_VEL
LIN {X 0,Y 136.821,Z 290.294,A -85,B 0,C 180,E1 -24975.781,E2 -24975.781} C_VEL
LIN {X 0,Y 136.6,Z 289.264,A -85,B 0,C 180,E1 -24976.013,E2 -24976.013} C_VEL
LIN {X 0,Y 136.098,Z 286.538,A -85,B 0,C 180,E1 -24981.704,E2 -24981.704} C_VEL
LIN {X 0,Y 136.054,Z 286.538,A -85,B 0,C 180,E1 -24985.738,E2 -24985.738} C_VEL
LIN {X 0,Y 136.047,Z 286.533,A -85,B 0,C 180,E1 -24989.202,E2 -24989.202} C_VEL
LIN {X 0,Y 135.349,Z 286.623,A -85,B 0,C 180,E1 -24991.676,E2 -24991.676} C_VEL
LIN {X 0,Y 133.782,Z 286.82,A -85,B 0,C 180,E1 -24994.118,E2 -24994.118} C_VEL
LIN {X 0,Y 129.381,Z 287.366,A -85,B 0,C 180,E1 -25000.855,E2 -25000.855} C_VEL
LIN {X 0,Y 129.105,Z 287.395,A -85,B 0,C 180,E1 -25002.632,E2 -25002.632} C_VEL
LIN {X 0,Y 129.375,Z 287.363,A -85,B 0,C 180,E1 -25007.901,E2 -25007.901} C_VEL
LIN {X 0,Y 129.472,Z 287.355,A -85,B 0,C 180,E1 -25010.624,E2 -25010.624} C_VEL
LIN {X 0,Y 130.085,Z 287.238,A -85,B 0,C 180,E1 -25019.996,E2 -25019.996} C_VEL
LIN {X 0,Y 129.513,Z 287.343,A -85,B 0,C 180,E1 -25029.365,E2 -25029.365} C_VEL
LIN {X 0,Y 129.389,Z 287.367,A -85,B 0,C 180,E1 -25032.545,E2 -25032.545} C_VEL
LIN {X 0,Y 129.148,Z 287.395,A -85,B 0,C 180,E1 -25039.053,E2 -25039.053} C_VEL
LIN {X 0,Y 129.103,Z 287.396,A -85,B 0,C 180,E1 -25042.395,E2 -25042.395} C_VEL
LIN {X 0,Y 129.023,Z 287.409,A -85,B 0,C 180,E1 -25045.83,E2 -25045.83} C_VEL
LIN {X 0,Y 129.01,Z 287.404,A -85,B 0,C 180,E1 -25049.355,E2 -25049.355} C_VEL
LIN {X 0,Y 129.018,Z 287.406,A -85,B 0,C 180,E1 -25055.207,E2 -25055.207} C_VEL
LIN {X 0,Y 128.999,Z 287.411,A -85,B 0,C 180,E1 -25060.821,E2 -25060.821} C_VEL
LIN {X 0,Y 128.964,Z 287.42,A -85,B 0,C 180,E1 -25065.103,E2 -25065.103} C_VEL
LIN {X 0,Y 128.977,Z 287.418,A -85,B 0,C 180,E1 -25069.711,E2 -25069.711} C_VEL
LIN {X 0,Y 128.974,Z 287.43,A -85,B 0,C 180,E1 -25074.612,E2 -25074.612} C_VEL
LIN {X 0,Y 130.016,Z 290.228,A -85,B 0,C 180,E1 -25075.365,E2 -25075.365} C_VEL
LIN {X 0,Y 131.693,Z 292.497,A -85,B 0,C 180,E1 -25076.338,E2 -25076.338} C_VEL
LIN {X 0,Y 137.134,Z 302.607,A -85,B 0,C 180,E1 -25079.836,E2 -25079.836} C_VEL
LIN {X 0,Y 138.546,Z 305.643,A -85,B 0,C 180,E1 -25080.825,E2 -25080.825} C_VEL
LIN {X 0,Y 140.674,Z 315.891,A -85,B 0,C 180,E1 -25083.574,E2 -25083.574} C_VEL
LIN {X 0,Y 141.601,Z 324.915,A -85,B 0,C 180,E1 -25086.078,E2 -25086.078} C_VEL
LIN {X 0,Y 141.875,Z 334.421,A -85,B 0,C 180,E1 -25088.953,E2 -25088.953} C_VEL
LIN {X 0,Y 141.573,Z 336.815,A -85,B 0,C 180,E1 -25089.666,E2 -25089.666} C_VEL
LIN {X 0,Y 138.658,Z 345.651,A -85,B 0,C 180,E1 -25092.295,E2 -25092.295} C_VEL
LIN {X 0,Y 135.62,Z 354.712,A -85,B 0,C 180,E1 -25095.75,E2 -25095.75} C_VEL
LIN {X 0,Y 132.439,Z 363.572,A -85,B 0,C 180,E1 -25100.069,E2 -25100.069} C_VEL
LIN {X 0,Y 129.875,Z 370.683,A -85,B 0,C 180,E1 -25104.566,E2 -25104.566} C_VEL
LIN {X 0,Y 128.388,Z 375.493,A -85,B 0,C 180,E1 -25108.432,E2 -25108.432} C_VEL
LIN {X 0,Y 127.148,Z 380.158,A -85,B 0,C 180,E1 -25113.168,E2 -25113.168} C_VEL
LIN {X 0,Y 126.289,Z 383.735,A -85,B 0,C 180,E1 -25117.997,E2 -25117.997} C_VEL
LIN {X 0,Y 125.968,Z 386.294,A -85,B 0,C 180,E1 -25122.895,E2 -25122.895} C_VEL
LIN {X 0,Y 126.175,Z 387.464,A -85,B 0,C 180,E1 -25126.17,E2 -25126.17} C_VEL
LIN {X 0,Y 126.607,Z 388.202,A -85,B 0,C 180,E1 -25129.454,E2 -25129.454} C_VEL
LIN {X 0,Y 127.287,Z 388.546,A -85,B 0,C 180,E1 -25132.736,E2 -25132.736} C_VEL
LIN {X 0,Y 128.337,Z 388.488,A -85,B 0,C 180,E1 -25135.982,E2 -25135.982} C_VEL
LIN {X 0,Y 130.431,Z 387.647,A -85,B 0,C 180,E1 -25140.452,E2 -25140.452} C_VEL
LIN {X 0,Y 133.587,Z 385.69,A -85,B 0,C 180,E1 -25145.359,E2 -25145.359} C_VEL
LIN {X 0,Y 137.556,Z 382.631,A -85,B 0,C 180,E1 -25149.976,E2 -25149.976} C_VEL
LIN {X 0,Y 141.86,Z 378.802,A -85,B 0,C 180,E1 -25153.913,E2 -25153.913} C_VEL
LIN {X 0,Y 147.682,Z 372.884,A -85,B 0,C 180,E1 -25158.227,E2 -25158.227} C_VEL
LIN {X 0,Y 153.85,Z 365.671,A -85,B 0,C 180,E1 -25161.997,E2 -25161.997} C_VEL
LIN {X 0,Y 158.37,Z 359.784,A -85,B 0,C 180,E1 -25164.328,E2 -25164.328} C_VEL
LIN {X 0,Y 159.684,Z 355.078,A -85,B 0,C 180,E1 -25166.741,E2 -25166.741} C_VEL
LIN {X 0,Y 160.501,Z 349.279,A -85,B 0,C 180,E1 -25169.769,E2 -25169.769} C_VEL
LIN {X 0,Y 160.407,Z 344.704,A -85,B 0,C 180,E1 -25172.35,E2 -25172.35} C_VEL
LIN {X 0,Y 159.564,Z 338.913,A -85,B 0,C 180,E1 -25175.961,E2 -25175.961} C_VEL
LIN {X 0,Y 158.034,Z 332.425,A -85,B 0,C 180,E1 -25180.52,E2 -25180.52} C_VEL
LIN {X 0,Y 157.026,Z 329.217,A -85,B 0,C 180,E1 -25183.09,E2 -25183.09} C_VEL
LIN {X 0,Y 155.479,Z 325.134,A -85,B 0,C 180,E1 -25186.941,E2 -25186.941} C_VEL
LIN {X 0,Y 154.624,Z 322.643,A -85,B 0,C 180,E1 -25189.528,E2 -25189.528} C_VEL
LIN {X 0,Y 153.106,Z 318.913,A -85,B 0,C 180,E1 -25194.736,E2 -25194.736} C_VEL
LIN {X 0,Y 151.883,Z 316.921,A -85,B 0,C 180,E1 -25200.003,E2 -25200.003} C_VEL
LIN {X 0,Y 151.487,Z 316.529,A -85,B 0,C 180,E1 -25202.662,E2 -25202.662} C_VEL
LIN {X 0,Y 151.25,Z 316.781,A -85,B 0,C 180,E1 -25208.016,E2 -25208.016} C_VEL
LIN {X 0,Y 152.349,Z 319.68,A -85,B 0,C 180,E1 -25216.072,E2 -25216.072} C_VEL
LIN {X 0,Y 153.077,Z 321.299,A -85,B 0,C 180,E1 -25218.75,E2 -25218.75} C_VEL
LIN {X 0,Y 154.745,Z 326.045,A -85,B 0,C 180,E1 -25224.13,E2 -25224.13} C_VEL
LIN {X 0,Y 156.409,Z 331.256,A -85,B 0,C 180,E1 -25228.633,E2 -25228.633} C_VEL
LIN {X 0,Y 157.761,Z 336.355,A -85,B 0,C 180,E1 -25232.319,E2 -25232.319} C_VEL
LIN {X 0,Y 159,Z 342.468,A -85,B 0,C 180,E1 -25236.205,E2 -25236.205} C_VEL
LIN {X 0,Y 159.788,Z 348.492,A -85,B 0,C 180,E1 -25239.697,E2 -25239.697} C_VEL
LIN {X 0,Y 159.691,Z 352.218,A -85,B 0,C 180,E1 -25241.569,E2 -25241.569} C_VEL
LIN {X 0,Y 158.28,Z 359.194,A -85,B 0,C 180,E1 -25244.731,E2 -25244.731} C_VEL
LIN {X 0,Y 155.819,Z 366.72,A -85,B 0,C 180,E1 -25248.298,E2 -25248.298} C_VEL
LIN {X 0,Y 155.225,Z 368.077,A -85,B 0,C 180,E1 -25248.967,E2 -25248.967} C_VEL
LIN {X 0,Y 149.277,Z 375.504,A -85,B 0,C 180,E1 -25252.264,E2 -25252.264} C_VEL
LIN {X 0,Y 143.904,Z 381.498,A -85,B 0,C 180,E1 -25255.832,E2 -25255.832} C_VEL
LIN {X 0,Y 139.311,Z 386.265,A -85,B 0,C 180,E1 -25259.704,E2 -25259.704} C_VEL
LIN {X 0,Y 135.159,Z 389.951,A -85,B 0,C 180,E1 -25263.77,E2 -25263.77} C_VEL
LIN {X 0,Y 131.776,Z 392.653,A -85,B 0,C 180,E1 -25268.08,E2 -25268.08} C_VEL
LIN {X 0,Y 128.586,Z 394.854,A -85,B 0,C 180,E1 -25274.141,E2 -25274.141} C_VEL
LIN {X 0,Y 126.866,Z 395.451,A -85,B 0,C 180,E1 -25280.434,E2 -25280.434} C_VEL
LIN {X 0,Y 126.385,Z 394.52,A -85,B 0,C 180,E1 -25286.812,E2 -25286.812} C_VEL
LIN {X 0,Y 126.511,Z 393.459,A -85,B 0,C 180,E1 -25290,E2 -25290} C_VEL
LIN {X 0,Y 126.387,Z 391.926,A -85,B 0,C 180,E1 -25293.188,E2 -25293.188} C_VEL
LIN {X 0,Y 126.654,Z 388.824,A -85,B 0,C 180,E1 -25297.974,E2 -25297.974} C_VEL
LIN {X 0,Y 127.411,Z 384.63,A -85,B 0,C 180,E1 -25302.746,E2 -25302.746} C_VEL
LIN {X 0,Y 129.181,Z 378.212,A -85,B 0,C 180,E1 -25308.229,E2 -25308.229} C_VEL
LIN {X 0,Y 131.648,Z 371.21,A -85,B 0,C 180,E1 -25312.77,E2 -25312.77} C_VEL
LIN {X 0,Y 133.809,Z 364.59,A -85,B 0,C 180,E1 -25316.197,E2 -25316.197} C_VEL
LIN {X 0,Y 137.175,Z 355.314,A -85,B 0,C 180,E1 -25319.968,E2 -25319.968} C_VEL
LIN {X 0,Y 138.677,Z 350.199,A -85,B 0,C 180,E1 -25321.721,E2 -25321.721} C_VEL
LIN {X 0,Y 139.657,Z 339.994,A -85,B 0,C 180,E1 -25325.033,E2 -25325.033} C_VEL
LIN {X 0,Y 140.004,Z 329.111,A -85,B 0,C 180,E1 -25328.058,E2 -25328.058} C_VEL
LIN {X 0,Y 139.398,Z 317.733,A -85,B 0,C 180,E1 -25330.86,E2 -25330.86} C_VEL
LIN {X 0,Y 138.012,Z 308.814,A -85,B 0,C 180,E1 -25332.938,E2 -25332.938} C_VEL
LIN {X 0,Y 134.528,Z 300.178,A -85,B 0,C 180,E1 -25335.423,E2 -25335.423} C_VEL
LIN {X 0,Y 131.409,Z 293.622,A -85,B 0,C 180,E1 -25337.395,E2 -25337.395} C_VEL
LIN {X 0,Y 129.594,Z 290.228,A -85,B 0,C 180,E1 -25338.494,E2 -25338.494} C_VEL
LIN {X 0,Y 129.309,Z 289.018,A -85,B 0,C 180,E1 -25338.772,E2 -25338.772} C_VEL
LIN {X 0,Y 128.987,Z 287.423,A -85,B 0,C 180,E1 -25342.684,E2 -25342.684} C_VEL
LIN {X 0,Y 128.974,Z 287.42,A -85,B 0,C 180,E1 -25346.977,E2 -25346.977} C_VEL
LIN {X 0,Y 129.019,Z 287.406,A -85,B 0,C 180,E1 -25350.639,E2 -25350.639} C_VEL
LIN {X 0,Y 129.109,Z 287.4,A -85,B 0,C 180,E1 -25357.598,E2 -25357.598} C_VEL
LIN {X 0,Y 129.105,Z 287.395,A -85,B 0,C 180,E1 -25362.632,E2 -25362.632} C_VEL
LIN {X 0,Y 128.489,Z 287.482,A -85,B 0,C 180,E1 -25365.239,E2 -25365.239} C_VEL
LIN {X 0,Y 126.979,Z 287.673,A -85,B 0,C 180,E1 -25367.817,E2 -25367.817} C_VEL
LIN {X 0,Y 122.776,Z 288.181,A -85,B 0,C 180,E1 -25374.942,E2 -25374.942} C_VEL
LIN {X 0,Y 122.6,Z 288.181,A -85,B 0,C 180,E1 -25376.817,E2 -25376.817} C_VEL
LIN {X 0,Y 123.039,Z 288.114,A -85,B 0,C 180,E1 -25379.996,E2 -25379.996} C_VEL
LIN {X 0,Y 122.413,Z 288.231,A -85,B 0,C 180,E1 -25387.17,E2 -25387.17} C_VEL
LIN {X 0,Y 122.36,Z 288.243,A -85,B 0,C 180,E1 -25392.469,E2 -25392.469} C_VEL
LIN {X 0,Y 122.04,Z 288.282,A -85,B 0,C 180,E1 -25400.209,E2 -25400.209} C_VEL
LIN {X 0,Y 121.977,Z 288.278,A -85,B 0,C 180,E1 -25403.781,E2 -25403.781} C_VEL
LIN {X 0,Y 121.923,Z 288.284,A -85,B 0,C 180,E1 -25410.16,E2 -25410.16} C_VEL
LIN {X 0,Y 121.93,Z 288.284,A -85,B 0,C 180,E1 -25416.202,E2 -25416.202} C_VEL
LIN {X 0,Y 121.923,Z 288.289,A -85,B 0,C 180,E1 -25421.467,E2 -25421.467} C_VEL
LIN {X 0,Y 121.904,Z 288.292,A -85,B 0,C 180,E1 -25428.538,E2 -25428.538} C_VEL
LIN {X 0,Y 121.863,Z 288.301,A -85,B 0,C 180,E1 -25431.516,E2 -25431.516} C_VEL
LIN {X 0,Y 122.884,Z 291.149,A -85,B 0,C 180,E1 -25432.426,E2 -25432.426} C_VEL
LIN {X 0,Y 124.724,Z 293.471,A -85,B 0,C 180,E1 -25433.623,E2 -25433.623} C_VEL
LIN {X 0,Y 126.693,Z 296.744,A -85,B 0,C 180,E1 -25434.98,E2 -25434.98} C_VEL
LIN {X 0,Y 131.638,Z 306.368,A -85,B 0,C 180,E1 -25438.666,E2 -25438.666} C_VEL
LIN {X 0,Y 132.875,Z 309.078,A -85,B 0,C 180,E1 -25439.676,E2 -25439.676} C_VEL
LIN {X 0,Y 134.409,Z 316.748,A -85,B 0,C 180,E1 -25441.928,E2 -25441.928} C_VEL
LIN {X 0,Y 135.245,Z 325.368,A -85,B 0,C 180,E1 -25444.499,E2 -25444.499} C_VEL
LIN {X 0,Y 135.438,Z 334.724,A -85,B 0,C 180,E1 -25447.5,E2 -25447.5} C_VEL
LIN {X 0,Y 135.326,Z 337.062,A -85,B 0,C 180,E1 -25448.283,E2 -25448.283} C_VEL
LIN {X 0,Y 131.946,Z 346.861,A -85,B 0,C 180,E1 -25451.362,E2 -25451.362} C_VEL
LIN {X 0,Y 128.701,Z 355.767,A -85,B 0,C 180,E1 -25454.967,E2 -25454.967} C_VEL
LIN {X 0,Y 125.397,Z 364.467,A -85,B 0,C 180,E1 -25459.505,E2 -25459.505} C_VEL
LIN {X 0,Y 122.81,Z 371.407,A -85,B 0,C 180,E1 -25464.252,E2 -25464.252} C_VEL
LIN {X 0,Y 120.75,Z 377.781,A -85,B 0,C 180,E1 -25470,E2 -25470} C_VEL
LIN {X 0,Y 119.801,Z 381.4,A -85,B 0,C 180,E1 -25474.285,E2 -25474.285} C_VEL
LIN {X 0,Y 118.955,Z 385.12,A -85,B 0,C 180,E1 -25480.209,E2 -25480.209} C_VEL
LIN {X 0,Y 118.883,Z 386.682,A -85,B 0,C 180,E1 -25483.678,E2 -25483.678} C_VEL
LIN {X 0,Y 119.567,Z 388.361,A -85,B 0,C 180,E1 -25489.884,E2 -25489.884} C_VEL
LIN {X 0,Y 120.526,Z 388.774,A -85,B 0,C 180,E1 -25494.09,E2 -25494.09} C_VEL
LIN {X 0,Y 121.756,Z 388.642,A -85,B 0,C 180,E1 -25497.501,E2 -25497.501} C_VEL
LIN {X 0,Y 123.787,Z 387.884,A -85,B 0,C 180,E1 -25501.62,E2 -25501.62} C_VEL
LIN {X 0,Y 127.598,Z 385.697,A -85,B 0,C 180,E1 -25507.29,E2 -25507.29} C_VEL
LIN {X 0,Y 131.422,Z 382.939,A -85,B 0,C 180,E1 -25511.531,E2 -25511.531} C_VEL
LIN {X 0,Y 136.62,Z 378.615,A -85,B 0,C 180,E1 -25516.068,E2 -25516.068} C_VEL
LIN {X 0,Y 142.933,Z 372.489,A -85,B 0,C 180,E1 -25520.477,E2 -25520.477} C_VEL
LIN {X 0,Y 149.431,Z 365.227,A -85,B 0,C 180,E1 -25524.221,E2 -25524.221} C_VEL
LIN {X 0,Y 152.752,Z 361.072,A -85,B 0,C 180,E1 -25525.908,E2 -25525.908} C_VEL
LIN {X 0,Y 154.356,Z 355.201,A -85,B 0,C 180,E1 -25529.193,E2 -25529.193} C_VEL
LIN {X 0,Y 154.952,Z 350.406,A -85,B 0,C 180,E1 -25532.012,E2 -25532.012} C_VEL
LIN {X 0,Y 154.6,Z 344.588,A -85,B 0,C 180,E1 -25535.853,E2 -25535.853} C_VEL
LIN {X 0,Y 153.733,Z 338.994,A -85,B 0,C 180,E1 -25539.952,E2 -25539.952} C_VEL
LIN {X 0,Y 152.584,Z 334.294,A -85,B 0,C 180,E1 -25543.96,E2 -25543.96} C_VEL
LIN {X 0,Y 151.371,Z 330.39,A -85,B 0,C 180,E1 -25547.944,E2 -25547.944} C_VEL
LIN {X 0,Y 150.335,Z 327.201,A -85,B 0,C 180,E1 -25551.941,E2 -25551.941} C_VEL
LIN {X 0,Y 149.8,Z 325.409,A -85,B 0,C 180,E1 -25554.619,E2 -25554.619} C_VEL
LIN {X 0,Y 148.801,Z 323.349,A -85,B 0,C 180,E1 -25560.003,E2 -25560.003} C_VEL
LIN {X 0,Y 148.45,Z 322.94,A -85,B 0,C 180,E1 -25562.717,E2 -25562.717} C_VEL
LIN {X 0,Y 148.213,Z 323.266,A -85,B 0,C 180,E1 -25568.182,E2 -25568.182} C_VEL
LIN {X 0,Y 149.187,Z 326.299,A -85,B 0,C 180,E1 -25576.422,E2 -25576.422} C_VEL
LIN {X 0,Y 149.93,Z 329.142,A -85,B 0,C 180,E1 -25580.368,E2 -25580.368} C_VEL
LIN {X 0,Y 150.784,Z 331.591,A -85,B 0,C 180,E1 -25583.343,E2 -25583.343} C_VEL
LIN {X 0,Y 151.965,Z 336.076,A -85,B 0,C 180,E1 -25587.55,E2 -25587.55} C_VEL
LIN {X 0,Y 153.187,Z 342.083,A -85,B 0,C 180,E1 -25592.2,E2 -25592.2} C_VEL
LIN {X 0,Y 153.98,Z 348.353,A -85,B 0,C 180,E1 -25596.398,E2 -25596.398} C_VEL
LIN {X 0,Y 154.201,Z 353.706,A -85,B 0,C 180,E1 -25599.652,E2 -25599.652} C_VEL
LIN {X 0,Y 153.294,Z 358.495,A -85,B 0,C 180,E1 -25602.082,E2 -25602.082} C_VEL
LIN {X 0,Y 150.849,Z 365.718,A -85,B 0,C 180,E1 -25605.667,E2 -25605.667} C_VEL
LIN {X 0,Y 149.716,Z 368.445,A -85,B 0,C 180,E1 -25607.106,E2 -25607.106} C_VEL
LIN {X 0,Y 147.887,Z 371.06,A -85,B 0,C 180,E1 -25608.295,E2 -25608.295} C_VEL
LIN {X 0,Y 141.783,Z 377.872,A -85,B 0,C 180,E1 -25611.714,E2 -25611.714} C_VEL
LIN {X 0,Y 136.096,Z 383.647,A -85,B 0,C 180,E1 -25615.72,E2 -25615.72} C_VEL
LIN {X 0,Y 131.668,Z 387.668,A -85,B 0,C 180,E1 -25619.532,E2 -25619.532} C_VEL
LIN {X 0,Y 127.549,Z 390.951,A -85,B 0,C 180,E1 -25623.846,E2 -25623.846} C_VEL
LIN {X 0,Y 123.221,Z 393.857,A -85,B 0,C 180,E1 -25629.989,E2 -25629.989} C_VEL
LIN {X 0,Y 121.74,Z 394.72,A -85,B 0,C 180,E1 -25633.224,E2 -25633.224} C_VEL
LIN {X 0,Y 119.851,Z 395.235,A -85,B 0,C 180,E1 -25639.868,E2 -25639.868} C_VEL
LIN {X 0,Y 119.425,Z 394.927,A -85,B 0,C 180,E1 -25643.241,E2 -25643.241} C_VEL
LIN {X 0,Y 119.292,Z 394.239,A -85,B 0,C 180,E1 -25646.623,E2 -25646.623} C_VEL
LIN {X 0,Y 119.424,Z 393.116,A -85,B 0,C 180,E1 -25650,E2 -25650} C_VEL
LIN {X 0,Y 119.295,Z 391.548,A -85,B 0,C 180,E1 -25653.377,E2 -25653.377} C_VEL
LIN {X 0,Y 119.613,Z 388.377,A -85,B 0,C 180,E1 -25658.447,E2 -25658.447} C_VEL
LIN {X 0,Y 120.47,Z 384.108,A -85,B 0,C 180,E1 -25663.494,E2 -25663.494} C_VEL
LIN {X 0,Y 122.405,Z 377.607,A -85,B 0,C 180,E1 -25669.277,E2 -25669.277} C_VEL
LIN {X 0,Y 125.044,Z 370.472,A -85,B 0,C 180,E1 -25674.046,E2 -25674.046} C_VEL
LIN {X 0,Y 128.028,Z 362.039,A -85,B 0,C 180,E1 -25678.42,E2 -25678.42} C_VEL
LIN {X 0,Y 131.029,Z 354.333,A -85,B 0,C 180,E1 -25681.53,E2 -25681.53} C_VEL
LIN {X 0,Y 132.129,Z 350.198,A -85,B 0,C 180,E1 -25683.038,E2 -25683.038} C_VEL
LIN {X 0,Y 133.306,Z 339.635,A -85,B 0,C 180,E1 -25686.632,E2 -25686.632} C_VEL
LIN {X 0,Y 133.722,Z 329.304,A -85,B 0,C 180,E1 -25689.662,E2 -25689.662} C_VEL
LIN {X 0,Y 133.196,Z 317.842,A -85,B 0,C 180,E1 -25692.682,E2 -25692.682} C_VEL
LIN {X 0,Y 132.347,Z 311.948,A -85,B 0,C 180,E1 -25694.195,E2 -25694.195} C_VEL
LIN {X 0,Y 128.702,Z 302.446,A -85,B 0,C 180,E1 -25697.216,E2 -25697.216} C_VEL
LIN {X 0,Y 126.176,Z 297.331,A -85,B 0,C 180,E1 -25699.015,E2 -25699.015} C_VEL
LIN {X 0,Y 124.292,Z 293.485,A -85,B 0,C 180,E1 -25700.348,E2 -25700.348} C_VEL
LIN {X 0,Y 122.545,Z 290.419,A -85,B 0,C 180,E1 -25701.536,E2 -25701.536} C_VEL
LIN {X 0,Y 122.047,Z 288.755,A -85,B 0,C 180,E1 -25702.003,E2 -25702.003} C_VEL
LIN {X 0,Y 121.911,Z 288.303,A -85,B 0,C 180,E1 -25703.81,E2 -25703.81} C_VEL
LIN {X 0,Y 121.928,Z 288.29,A -85,B 0,C 180,E1 -25709.836,E2 -25709.836} C_VEL
LIN {X 0,Y 121.982,Z 288.282,A -85,B 0,C 180,E1 -25716.211,E2 -25716.211} C_VEL
LIN {X 0,Y 122.033,Z 288.286,A -85,B 0,C 180,E1 -25719.781,E2 -25719.781} C_VEL
LIN {X 0,Y 122.237,Z 288.259,A -85,B 0,C 180,E1 -25726.7,E2 -25726.7} C_VEL
LIN {X 0,Y 122.405,Z 288.232,A -85,B 0,C 180,E1 -25730.078,E2 -25730.078} C_VEL
LIN {X 0,Y 122.6,Z 288.181,A -85,B 0,C 180,E1 -25736.817,E2 -25736.817} C_VEL
LIN {X 0,Y 122.389,Z 288.198,A -85,B 0,C 180,E1 -25738.647,E2 -25738.647} C_VEL
LIN {X 0,Y 121.092,Z 288.374,A -85,B 0,C 180,E1 -25741.36,E2 -25741.36} C_VEL
LIN {X 0,Y 115.679,Z 289.067,A -85,B 0,C 180,E1 -25749.753,E2 -25749.753} C_VEL
LIN {X 0,Y 115.295,Z 289.116,A -85,B 0,C 180,E1 -25751.754,E2 -25751.754} C_VEL
LIN {X 0,Y 115.007,Z 289.149,A -85,B 0,C 180,E1 -25757.787,E2 -25757.787} C_VEL
LIN {X 0,Y 114.942,Z 289.155,A -85,B 0,C 180,E1 -25763.489,E2 -25763.489} C_VEL
LIN {X 0,Y 114.858,Z 289.165,A -85,B 0,C 180,E1 -25771.06,E2 -25771.06} C_VEL
LIN {X 0,Y 114.841,Z 289.169,A -85,B 0,C 180,E1 -25777.727,E2 -25777.727} C_VEL
LIN {X 0,Y 114.833,Z 289.169,A -85,B 0,C 180,E1 -25782.743,E2 -25782.743} C_VEL
LIN {X 0,Y 114.852,Z 289.169,A -85,B 0,C 180,E1 -25787.929,E2 -25787.929} C_VEL
LIN {X 0,Y 115.893,Z 292.103,A -85,B 0,C 180,E1 -25789.032,E2 -25789.032} C_VEL
LIN {X 0,Y 117.768,Z 294.408,A -85,B 0,C 180,E1 -25790.447,E2 -25790.447} C_VEL
LIN {X 0,Y 119.778,Z 297.81,A -85,B 0,C 180,E1 -25792.081,E2 -25792.081} C_VEL
LIN {X 0,Y 123.931,Z 305.163,A -85,B 0,C 180,E1 -25795.453,E2 -25795.453} C_VEL
LIN {X 0,Y 127.485,Z 313.242,A -85,B 0,C 180,E1 -25798.732,E2 -25798.732} C_VEL
LIN {X 0,Y 128.813,Z 322.501,A -85,B 0,C 180,E1 -25801.697,E2 -25801.697} C_VEL
LIN {X 0,Y 129.131,Z 332.609,A -85,B 0,C 180,E1 -25805.052,E2 -25805.052} C_VEL
LIN {X 0,Y 129.007,Z 337.316,A -85,B 0,C 180,E1 -25806.737,E2 -25806.737} C_VEL
LIN {X 0,Y 125.937,Z 346.108,A -85,B 0,C 180,E1 -25809.587,E2 -25809.587} C_VEL
LIN {X 0,Y 122.53,Z 355.161,A -85,B 0,C 180,E1 -25813.335,E2 -25813.335} C_VEL
LIN {X 0,Y 118.963,Z 364.014,A -85,B 0,C 180,E1 -25818.067,E2 -25818.067} C_VEL
LIN {X 0,Y 116.094,Z 371.113,A -85,B 0,C 180,E1 -25823.046,E2 -25823.046} C_VEL
LIN {X 0,Y 114.087,Z 376.771,A -85,B 0,C 180,E1 -25828.235,E2 -25828.235} C_VEL
LIN {X 0,Y 112.722,Z 381.581,A -85,B 0,C 180,E1 -25834.067,E2 -25834.067} C_VEL
LIN {X 0,Y 111.807,Z 385.558,A -85,B 0,C 180,E1 -25840.869,E2 -25840.869} C_VEL
LIN {X 0,Y 111.826,Z 387.037,A -85,B 0,C 180,E1 -25844.559,E2 -25844.559} C_VEL
LIN {X 0,Y 112.559,Z 388.543,A -85,B 0,C 180,E1 -25850.529,E2 -25850.529} C_VEL
LIN {X 0,Y 113.828,Z 388.993,A -85,B 0,C 180,E1 -25855.606,E2 -25855.606} C_VEL
LIN {X 0,Y 115.25,Z 388.785,A -85,B 0,C 180,E1 -25859.198,E2 -25859.198} C_VEL
LIN {X 0,Y 117.196,Z 388.122,A -85,B 0,C 180,E1 -25862.916,E2 -25862.916} C_VEL
LIN {X 0,Y 119.234,Z 387.153,A -85,B 0,C 180,E1 -25866.115,E2 -25866.115} C_VEL
LIN {X 0,Y 121.769,Z 385.673,A -85,B 0,C 180,E1 -25869.409,E2 -25869.409} C_VEL
LIN {X 0,Y 125.421,Z 383.234,A -85,B 0,C 180,E1 -25873.249,E2 -25873.249} C_VEL
LIN {X 0,Y 131.577,Z 378.394,A -85,B 0,C 180,E1 -25878.398,E2 -25878.398} C_VEL
LIN {X 0,Y 138.004,Z 372.482,A -85,B 0,C 180,E1 -25882.651,E2 -25882.651} C_VEL
LIN {X 0,Y 144.097,Z 366.046,A -85,B 0,C 180,E1 -25886.008,E2 -25886.008} C_VEL
LIN {X 0,Y 146.4,Z 363.37,A -85,B 0,C 180,E1 -25887.148,E2 -25887.148} C_VEL
LIN {X 0,Y 147.153,Z 362.205,A -85,B 0,C 180,E1 -25887.732,E2 -25887.732} C_VEL
LIN {X 0,Y 148.818,Z 356.643,A -85,B 0,C 180,E1 -25891.149,E2 -25891.149} C_VEL
LIN {X 0,Y 149.305,Z 353.179,A -85,B 0,C 180,E1 -25893.423,E2 -25893.423} C_VEL
LIN {X 0,Y 149.29,Z 349.051,A -85,B 0,C 180,E1 -25896.416,E2 -25896.416} C_VEL
LIN {X 0,Y 148.74,Z 343.459,A -85,B 0,C 180,E1 -25900.906,E2 -25900.906} C_VEL
LIN {X 0,Y 147.975,Z 339.199,A -85,B 0,C 180,E1 -25904.861,E2 -25904.861} C_VEL
LIN {X 0,Y 146.843,Z 334.431,A -85,B 0,C 180,E1 -25910.36,E2 -25910.36} C_VEL
LIN {X 0,Y 146.134,Z 331.713,A -85,B 0,C 180,E1 -25914.484,E2 -25914.484} C_VEL
LIN {X 0,Y 145.713,Z 330.444,A -85,B 0,C 180,E1 -25917.239,E2 -25917.239} C_VEL
LIN {X 0,Y 145.368,Z 329.593,A -85,B 0,C 180,E1 -25920.003,E2 -25920.003} C_VEL
LIN {X 0,Y 145.068,Z 329.182,A -85,B 0,C 180,E1 -25922.78,E2 -25922.78} C_VEL
LIN {X 0,Y 144.82,Z 329.597,A -85,B 0,C 180,E1 -25928.375,E2 -25928.375} C_VEL
LIN {X 0,Y 145.226,Z 331.697,A -85,B 0,C 180,E1 -25934.57,E2 -25934.57} C_VEL
LIN {X 0,Y 145.58,Z 332.812,A -85,B 0,C 180,E1 -25936.841,E2 -25936.841} C_VEL
LIN {X 0,Y 146.59,Z 336.972,A -85,B 0,C 180,E1 -25942.557,E2 -25942.557} C_VEL
LIN {X 0,Y 147.448,Z 341.306,A -85,B 0,C 180,E1 -25946.927,E2 -25946.927} C_VEL
LIN {X 0,Y 148.208,Z 346.719,A -85,B 0,C 180,E1 -25951.444,E2 -25951.444} C_VEL
LIN {X 0,Y 148.549,Z 351.011,A -85,B 0,C 180,E1 -25954.596,E2 -25954.596} C_VEL
LIN {X 0,Y 148.546,Z 356.841,A -85,B 0,C 180,E1 -25958.534,E2 -25958.534} C_VEL
LIN {X 0,Y 147.376,Z 361.422,A -85,B 0,C 180,E1 -25961.062,E2 -25961.062} C_VEL
LIN {X 0,Y 144.311,Z 368.817,A -85,B 0,C 180,E1 -25965.079,E2 -25965.079} C_VEL
LIN {X 0,Y 143.651,Z 370.128,A -85,B 0,C 180,E1 -25965.801,E2 -25965.801} C_VEL
LIN {X 0,Y 137.291,Z 377.079,A -85,B 0,C 180,E1 -25969.258,E2 -25969.258} C_VEL
LIN {X 0,Y 130.602,Z 383.477,A -85,B 0,C 180,E1 -25973.707,E2 -25973.707} C_VEL
LIN {X 0,Y 125.6,Z 387.721,A -85,B 0,C 180,E1 -25977.889,E2 -25977.889} C_VEL
LIN {X 0,Y 121.182,Z 390.933,A -85,B 0,C 180,E1 -25982.358,E2 -25982.358} C_VEL
LIN {X 0,Y 116.547,Z 393.769,A -85,B 0,C 180,E1 -25988.789,E2 -25988.789} C_VEL
LIN {X 0,Y 113.699,Z 394.981,A -85,B 0,C 180,E1 -25995.686,E2 -25995.686} C_VEL
LIN {X 0,Y 112.357,Z 394.678,A -85,B 0,C 180,E1 -26002.814,E2 -26002.814} C_VEL
LIN {X 0,Y 112.21,Z 393.94,A -85,B 0,C 180,E1 -26006.409,E2 -26006.409} C_VEL
LIN {X 0,Y 112.339,Z 392.771,A -85,B 0,C 180,E1 -26010,E2 -26010} C_VEL
LIN {X 0,Y 112.247,Z 390.212,A -85,B 0,C 180,E1 -26015.389,E2 -26015.389} C_VEL
LIN {X 0,Y 112.804,Z 386.616,A -85,B 0,C 180,E1 -26020.772,E2 -26020.772} C_VEL
LIN {X 0,Y 114.015,Z 381.876,A -85,B 0,C 180,E1 -26026.104,E2 -26026.104} C_VEL
LIN {X 0,Y 116.623,Z 374.737,A -85,B 0,C 180,E1 -26032.125,E2 -26032.125} C_VEL
LIN {X 0,Y 119.673,Z 366.947,A -85,B 0,C 180,E1 -26037.073,E2 -26037.073} C_VEL
LIN {X 0,Y 121.959,Z 360.825,A -85,B 0,C 180,E1 -26040.18,E2 -26040.18} C_VEL
LIN {X 0,Y 125.313,Z 352.34,A -85,B 0,C 180,E1 -26043.629,E2 -26043.629} C_VEL
LIN {X 0,Y 126.687,Z 343.071,A -85,B 0,C 180,E1 -26047.105,E2 -26047.105} C_VEL
LIN {X 0,Y 127.463,Z 333.268,A -85,B 0,C 180,E1 -26050.296,E2 -26050.296} C_VEL
LIN {X 0,Y 127.418,Z 322.454,A -85,B 0,C 180,E1 -26053.448,E2 -26053.448} C_VEL
LIN {X 0,Y 126.932,Z 316.014,A -85,B 0,C 180,E1 -26055.201,E2 -26055.201} C_VEL
LIN {X 0,Y 123.984,Z 307.291,A -85,B 0,C 180,E1 -26058.233,E2 -26058.233} C_VEL
LIN {X 0,Y 119.943,Z 298.479,A -85,B 0,C 180,E1 -26061.625,E2 -26061.625} C_VEL
LIN {X 0,Y 118.032,Z 294.655,A -85,B 0,C 180,E1 -26063.195,E2 -26063.195} C_VEL
LIN {X 0,Y 117.502,Z 293.861,A -85,B 0,C 180,E1 -26063.582,E2 -26063.582} C_VEL
LIN {X 0,Y 115.573,Z 291.473,A -85,B 0,C 180,E1 -26064.973,E2 -26064.973} C_VEL
LIN {X 0,Y 114.833,Z 289.182,A -85,B 0,C 180,E1 -26065.781,E2 -26065.781} C_VEL
LIN {X 0,Y 114.858,Z 289.169,A -85,B 0,C 180,E1 -26070.687,E2 -26070.687} C_VEL
LIN {X 0,Y 114.947,Z 289.159,A -85,B 0,C 180,E1 -26076.506,E2 -26076.506} C_VEL
LIN {X 0,Y 115,Z 289.152,A -85,B 0,C 180,E1 -26082.204,E2 -26082.204} C_VEL
LIN {X 0,Y 115.255,Z 289.125,A -85,B 0,C 180,E1 -26087.324,E2 -26087.324} C_VEL
LIN {X 0,Y 115.363,Z 289.117,A -85,B 0,C 180,E1 -26092.997,E2 -26092.997} C_VEL
LIN {X 0,Y 115.99,Z 288.99,A -85,B 0,C 180,E1 -26099.996,E2 -26099.996} C_VEL
LIN {X 0,Y 115.381,Z 289.113,A -85,B 0,C 180,E1 -26107.061,E2 -26107.061} C_VEL
LIN {X 0,Y 115.295,Z 289.116,A -85,B 0,C 180,E1 -26111.754,E2 -26111.754} C_VEL
LIN {X 0,Y 114.542,Z 289.225,A -85,B 0,C 180,E1 -26114.664,E2 -26114.664} C_VEL
LIN {X 0,Y 112.889,Z 289.444,A -85,B 0,C 180,E1 -26117.536,E2 -26117.536} C_VEL
LIN {X 0,Y 108.115,Z 290.028,A -85,B 0,C 180,E1 -26125.523,E2 -26125.523} C_VEL
LIN {X 0,Y 107.723,Z 290.06,A -85,B 0,C 180,E1 -26127.656,E2 -26127.656} C_VEL
LIN {X 0,Y 107.79,Z 290.049,A -85,B 0,C 180,E1 -26132.049,E2 -26132.049} C_VEL
LIN {X 0,Y 107.744,Z 290.057,A -85,B 0,C 180,E1 -26138.489,E2 -26138.489} C_VEL
LIN {X 0,Y 107.762,Z 290.072,A -85,B 0,C 180,E1 -26143.512,E2 -26143.512} C_VEL
LIN {X 0,Y 108.586,Z 292.679,A -85,B 0,C 180,E1 -26144.607,E2 -26144.607} C_VEL
LIN {X 0,Y 110.753,Z 295.024,A -85,B 0,C 180,E1 -26146.527,E2 -26146.527} C_VEL
LIN {X 0,Y 112.835,Z 298.701,A -85,B 0,C 180,E1 -26148.583,E2 -26148.583} C_VEL
LIN {X 0,Y 113.918,Z 300.481,A -85,B 0,C 180,E1 -26149.592,E2 -26149.592} C_VEL
LIN {X 0,Y 118.012,Z 307.86,A -85,B 0,C 180,E1 -26153.45,E2 -26153.45} C_VEL
LIN {X 0,Y 121.547,Z 315.797,A -85,B 0,C 180,E1 -26157.121,E2 -26157.121} C_VEL
LIN {X 0,Y 122.236,Z 318.852,A -85,B 0,C 180,E1 -26158.278,E2 -26158.278} C_VEL
LIN {X 0,Y 122.915,Z 328.268,A -85,B 0,C 180,E1 -26161.563,E2 -26161.563} C_VEL
LIN {X 0,Y 122.619,Z 338.689,A -85,B 0,C 180,E1 -26165.447,E2 -26165.447} C_VEL
LIN {X 0,Y 119.343,Z 347.295,A -85,B 0,C 180,E1 -26168.404,E2 -26168.404} C_VEL
LIN {X 0,Y 115.703,Z 356.196,A -85,B 0,C 180,E1 -26172.32,E2 -26172.32} C_VEL
LIN {X 0,Y 112.581,Z 363.544,A -85,B 0,C 180,E1 -26176.462,E2 -26176.462} C_VEL
LIN {X 0,Y 109.423,Z 370.796,A -85,B 0,C 180,E1 -26181.691,E2 -26181.691} C_VEL
LIN {X 0,Y 107.568,Z 375.674,A -85,B 0,C 180,E1 -26186.254,E2 -26186.254} C_VEL
LIN {X 0,Y 106.02,Z 380.429,A -85,B 0,C 180,E1 -26191.899,E2 -26191.899} C_VEL
LIN {X 0,Y 104.999,Z 384.09,A -85,B 0,C 180,E1 -26197.693,E2 -26197.693} C_VEL
LIN {X 0,Y 104.694,Z 385.977,A -85,B 0,C 180,E1 -26201.618,E2 -26201.618} C_VEL
LIN {X 0,Y 104.777,Z 387.389,A -85,B 0,C 180,E1 -26205.563,E2 -26205.563} C_VEL
LIN {X 0,Y 105.587,Z 388.727,A -85,B 0,C 180,E1 -26211.288,E2 -26211.288} C_VEL
LIN {X 0,Y 107.223,Z 389.183,A -85,B 0,C 180,E1 -26217.31,E2 -26217.31} C_VEL
LIN {X 0,Y 110.635,Z 388.369,A -85,B 0,C 180,E1 -26224.337,E2 -26224.337} C_VEL
LIN {X 0,Y 113.32,Z 387.199,A -85,B 0,C 180,E1 -26228.329,E2 -26228.329} C_VEL
LIN {X 0,Y 116.144,Z 385.643,A -85,B 0,C 180,E1 -26231.729,E2 -26231.729} C_VEL
LIN {X 0,Y 120.926,Z 382.602,A -85,B 0,C 180,E1 -26236.348,E2 -26236.348} C_VEL
LIN {X 0,Y 126.785,Z 378.178,A -85,B 0,C 180,E1 -26240.899,E2 -26240.899} C_VEL
LIN {X 0,Y 133.066,Z 372.709,A -85,B 0,C 180,E1 -26244.838,E2 -26244.838} C_VEL
LIN {X 0,Y 140.087,Z 365.619,A -85,B 0,C 180,E1 -26248.523,E2 -26248.523} C_VEL
LIN {X 0,Y 141.031,Z 364.585,A -85,B 0,C 180,E1 -26248.96,E2 -26248.96} C_VEL
LIN {X 0,Y 142.574,Z 360.979,A -85,B 0,C 180,E1 -26251.299,E2 -26251.299} C_VEL
LIN {X 0,Y 143.505,Z 357.328,A -85,B 0,C 180,E1 -26253.851,E2 -26253.851} C_VEL
LIN {X 0,Y 143.809,Z 351.897,A -85,B 0,C 180,E1 -26258.204,E2 -26258.204} C_VEL
LIN {X 0,Y 143.568,Z 346.692,A -85,B 0,C 180,E1 -26262.923,E2 -26262.923} C_VEL
LIN {X 0,Y 143.007,Z 342.721,A -85,B 0,C 180,E1 -26267.227,E2 -26267.227} C_VEL
LIN {X 0,Y 142.439,Z 339.523,A -85,B 0,C 180,E1 -26271.491,E2 -26271.491} C_VEL
LIN {X 0,Y 142.144,Z 337.786,A -85,B 0,C 180,E1 -26274.328,E2 -26274.328} C_VEL
LIN {X 0,Y 141.834,Z 336.471,A -85,B 0,C 180,E1 -26277.163,E2 -26277.163} C_VEL
LIN {X 0,Y 141.562,Z 335.61,A -85,B 0,C 180,E1 -26280.003,E2 -26280.003} C_VEL
LIN {X 0,Y 141.331,Z 335.201,A -85,B 0,C 180,E1 -26282.854,E2 -26282.854} C_VEL
LIN {X 0,Y 141.05,Z 335.722,A -85,B 0,C 180,E1 -26288.6,E2 -26288.6} C_VEL
LIN {X 0,Y 141.309,Z 337.629,A -85,B 0,C 180,E1 -26294.403,E2 -26294.403} C_VEL
LIN {X 0,Y 141.606,Z 339.154,A -85,B 0,C 180,E1 -26297.328,E2 -26297.328} C_VEL
LIN {X 0,Y 142.153,Z 342.2,A -85,B 0,C 180,E1 -26301.768,E2 -26301.768} C_VEL
LIN {X 0,Y 142.698,Z 346.344,A -85,B 0,C 180,E1 -26306.315,E2 -26306.315} C_VEL
LIN {X 0,Y 143.035,Z 350.953,A -85,B 0,C 180,E1 -26310.47,E2 -26310.47} C_VEL
LIN {X 0,Y 143.088,Z 355.863,A -85,B 0,C 180,E1 -26314.393,E2 -26314.393} C_VEL
LIN {X 0,Y 142.951,Z 359.086,A -85,B 0,C 180,E1 -26316.785,E2 -26316.785} C_VEL
LIN {X 0,Y 142.211,Z 362.205,A -85,B 0,C 180,E1 -26318.785,E2 -26318.785} C_VEL
LIN {X 0,Y 139.722,Z 367.913,A -85,B 0,C 180,E1 -26322.106,E2 -26322.106} C_VEL
LIN {X 0,Y 137.588,Z 371.682,A -85,B 0,C 180,E1 -26324.348,E2 -26324.348} C_VEL
LIN {X 0,Y 130.923,Z 378.303,A -85,B 0,C 180,E1 -26327.857,E2 -26327.857} C_VEL
LIN {X 0,Y 124.934,Z 383.609,A -85,B 0,C 180,E1 -26331.773,E2 -26331.773} C_VEL
LIN {X 0,Y 119.646,Z 387.774,A -85,B 0,C 180,E1 -26336.081,E2 -26336.081} C_VEL
LIN {X 0,Y 114.908,Z 390.915,A -85,B 0,C 180,E1 -26340.707,E2 -26340.707} C_VEL
LIN {X 0,Y 112.238,Z 392.495,A -85,B 0,C 180,E1 -26344.004,E2 -26344.004} C_VEL
LIN {X 0,Y 109.935,Z 393.665,A -85,B 0,C 180,E1 -26347.446,E2 -26347.446} C_VEL
LIN {X 0,Y 106.822,Z 394.797,A -85,B 0,C 180,E1 -26354.743,E2 -26354.743} C_VEL
LIN {X 0,Y 105.301,Z 394.425,A -85,B 0,C 180,E1 -26362.329,E2 -26362.329} C_VEL
LIN {X 0,Y 105.119,Z 393.625,A -85,B 0,C 180,E1 -26366.167,E2 -26366.167} C_VEL
LIN {X 0,Y 105.24,Z 392.423,A -85,B 0,C 180,E1 -26370,E2 -26370} C_VEL
LIN {X 0,Y 105.193,Z 389.795,A -85,B 0,C 180,E1 -26375.752,E2 -26375.752} C_VEL
LIN {X 0,Y 105.814,Z 386.123,A -85,B 0,C 180,E1 -26381.493,E2 -26381.493} C_VEL
LIN {X 0,Y 107.171,Z 381.302,A -85,B 0,C 180,E1 -26387.163,E2 -26387.163} C_VEL
LIN {X 0,Y 109.561,Z 375.206,A -85,B 0,C 180,E1 -26392.636,E2 -26392.636} C_VEL
LIN {X 0,Y 112.735,Z 367.592,A -85,B 0,C 180,E1 -26397.875,E2 -26397.875} C_VEL
LIN {X 0,Y 115.404,Z 360.903,A -85,B 0,C 180,E1 -26401.499,E2 -26401.499} C_VEL
LIN {X 0,Y 118.27,Z 354.304,A -85,B 0,C 180,E1 -26404.368,E2 -26404.368} C_VEL
LIN {X 0,Y 119.314,Z 350.16,A -85,B 0,C 180,E1 -26406.088,E2 -26406.088} C_VEL
LIN {X 0,Y 120.769,Z 340.387,A -85,B 0,C 180,E1 -26409.801,E2 -26409.801} C_VEL
LIN {X 0,Y 121.457,Z 330.991,A -85,B 0,C 180,E1 -26412.949,E2 -26412.949} C_VEL
LIN {X 0,Y 121.376,Z 321.131,A -85,B 0,C 180,E1 -26415.981,E2 -26415.981} C_VEL
LIN {X 0,Y 121.002,Z 318.078,A -85,B 0,C 180,E1 -26416.959,E2 -26416.959} C_VEL
LIN {X 0,Y 118.107,Z 309.563,A -85,B 0,C 180,E1 -26420.3,E2 -26420.3} C_VEL
LIN {X 0,Y 115.088,Z 302.593,A -85,B 0,C 180,E1 -26423.318,E2 -26423.318} C_VEL
LIN {X 0,Y 113.437,Z 299.246,A -85,B 0,C 180,E1 -26424.894,E2 -26424.894} C_VEL
LIN {X 0,Y 111.334,Z 295.932,A -85,B 0,C 180,E1 -26426.772,E2 -26426.772} C_VEL
LIN {X 0,Y 110.724,Z 294.977,A -85,B 0,C 180,E1 -26427.337,E2 -26427.337} C_VEL
LIN {X 0,Y 108.656,Z 292.627,A -85,B 0,C 180,E1 -26429.104,E2 -26429.104} C_VEL
LIN {X 0,Y 107.815,Z 290.046,A -85,B 0,C 180,E1 -26430.191,E2 -26430.191} C_VEL
LIN {X 0,Y 107.91,Z 290.036,A -85,B 0,C 180,E1 -26436.993,E2 -26436.993} C_VEL
LIN {X 0,Y 108.025,Z 290.031,A -85,B 0,C 180,E1 -26444.912,E2 -26444.912} C_VEL
LIN {X 0,Y 108.255,Z 289.991,A -85,B 0,C 180,E1 -26448.765,E2 -26448.765} C_VEL
LIN {X 0,Y 108.44,Z 289.946,A -85,B 0,C 180,E1 -26456.28,E2 -26456.28} C_VEL
LIN {X 0,Y 108.916,Z 289.87,A -85,B 0,C 180,E1 -26459.996,E2 -26459.996} C_VEL
LIN {X 0,Y 108.325,Z 289.989,A -85,B 0,C 180,E1 -26467.451,E2 -26467.451} C_VEL
LIN {X 0,Y 108.195,Z 290.008,A -85,B 0,C 180,E1 -26473.011,E2 -26473.011} C_VEL
LIN {X 0,Y 107.9,Z 290.041,A -85,B 0,C 180,E1 -26479.001,E2 -26479.001} C_VEL
LIN {X 0,Y 107.851,Z 290.037,A -85,B 0,C 180,E1 -26484.178,E2 -26484.178} C_VEL
LIN {X 0,Y 107.723,Z 290.06,A -85,B 0,C 180,E1 -26487.656,E2 -26487.656} C_VEL
LIN {X 0,Y 107.072,Z 290.305,A -85,B 0,C 180,E1 -26490.727,E2 -26490.727} C_VEL
LIN {X 0,Y 105.823,Z 291.075,A -85,B 0,C 180,E1 -26493.769,E2 -26493.769} C_VEL
LIN {X 0,Y 104.295,Z 292.998,A -85,B 0,C 180,E1 -26497.768,E2 -26497.768} C_VEL
LIN {X 0,Y 103.965,Z 295.233,A -85,B 0,C 180,E1 -26500.659,E2 -26500.659} C_VEL
LIN {X 0,Y 104.438,Z 297.139,A -85,B 0,C 180,E1 -26502.433,E2 -26502.433} C_VEL
LIN {X 0,Y 104.943,Z 298.218,A -85,B 0,C 180,E1 -26503.234,E2 -26503.234} C_VEL
LIN {X 0,Y 107.374,Z 301.586,A -85,B 0,C 180,E1 -26505.846,E2 -26505.846} C_VEL
LIN {X 0,Y 111.617,Z 309.352,A -85,B 0,C 180,E1 -26510.606,E2 -26510.606} C_VEL
LIN {X 0,Y 114.958,Z 316.743,A -85,B 0,C 180,E1 -26514.53,E2 -26514.53} C_VEL
LIN {X 0,Y 116.344,Z 320.544,A -85,B 0,C 180,E1 -26516.396,E2 -26516.396} C_VEL
LIN {X 0,Y 116.848,Z 329.783,A -85,B 0,C 180,E1 -26519.906,E2 -26519.906} C_VEL
LIN {X 0,Y 116.433,Z 338.957,A -85,B 0,C 180,E1 -26523.567,E2 -26523.567} C_VEL
LIN {X 0,Y 115.348,Z 342.326,A -85,B 0,C 180,E1 -26524.755,E2 -26524.755} C_VEL
LIN {X 0,Y 112.036,Z 350.384,A -85,B 0,C 180,E1 -26527.891,E2 -26527.891} C_VEL
LIN {X 0,Y 108.229,Z 358.767,A -85,B 0,C 180,E1 -26532.035,E2 -26532.035} C_VEL
LIN {X 0,Y 104.412,Z 366.966,A -85,B 0,C 180,E1 -26537.364,E2 -26537.364} C_VEL
LIN {X 0,Y 102.02,Z 372.538,A -85,B 0,C 180,E1 -26542.081,E2 -26542.081} C_VEL
LIN {X 0,Y 99.816,Z 377.998,A -85,B 0,C 180,E1 -26547.982,E2 -26547.982} C_VEL
LIN {X 0,Y 98.447,Z 382.279,A -85,B 0,C 180,E1 -26554.093,E2 -26554.093} C_VEL
LIN {X 0,Y 97.828,Z 384.569,A -85,B 0,C 180,E1 -26558.261,E2 -26558.261} C_VEL
LIN {X 0,Y 97.589,Z 386.371,A -85,B 0,C 180,E1 -26562.477,E2 -26562.477} C_VEL
LIN {X 0,Y 97.775,Z 387.741,A -85,B 0,C 180,E1 -26566.709,E2 -26566.709} C_VEL
LIN {X 0,Y 98.616,Z 388.909,A -85,B 0,C 180,E1 -26572.124,E2 -26572.124} C_VEL
LIN {X 0,Y 100.716,Z 389.369,A -85,B 0,C 180,E1 -26579.238,E2 -26579.238} C_VEL
LIN {X 0,Y 104.199,Z 388.607,A -85,B 0,C 180,E1 -26585.974,E2 -26585.974} C_VEL
LIN {X 0,Y 107.593,Z 387.22,A -85,B 0,C 180,E1 -26590.782,E2 -26590.782} C_VEL
LIN {X 0,Y 113.812,Z 383.832,A -85,B 0,C 180,E1 -26597.221,E2 -26597.221} C_VEL
LIN {X 0,Y 120.136,Z 379.591,A -85,B 0,C 180,E1 -26602.161,E2 -26602.161} C_VEL
LIN {X 0,Y 126.825,Z 374.283,A -85,B 0,C 180,E1 -26606.353,E2 -26606.353} C_VEL
LIN {X 0,Y 133.892,Z 367.724,A -85,B 0,C 180,E1 -26610.005,E2 -26610.005} C_VEL
LIN {X 0,Y 135.125,Z 366.459,A -85,B 0,C 180,E1 -26610.594,E2 -26610.594} C_VEL
LIN {X 0,Y 136.045,Z 365.13,A -85,B 0,C 180,E1 -26611.424,E2 -26611.424} C_VEL
LIN {X 0,Y 137.513,Z 361.331,A -85,B 0,C 180,E1 -26614.256,E2 -26614.256} C_VEL
LIN {X 0,Y 138.116,Z 357.825,A -85,B 0,C 180,E1 -26617.257,E2 -26617.257} C_VEL
LIN {X 0,Y 138.347,Z 354.13,A -85,B 0,C 180,E1 -26620.723,E2 -26620.723} C_VEL
LIN {X 0,Y 138.327,Z 349.764,A -85,B 0,C 180,E1 -26625.287,E2 -26625.287} C_VEL
LIN {X 0,Y 138.03,Z 346.172,A -85,B 0,C 180,E1 -26629.969,E2 -26629.969} C_VEL
LIN {X 0,Y 137.805,Z 343.621,A -85,B 0,C 180,E1 -26634.149,E2 -26634.149} C_VEL
LIN {X 0,Y 137.618,Z 342.302,A -85,B 0,C 180,E1 -26637.076,E2 -26637.076} C_VEL
LIN {X 0,Y 137.43,Z 341.418,A -85,B 0,C 180,E1 -26640.004,E2 -26640.004} C_VEL
LIN {X 0,Y 137.238,Z 341.019,A -85,B 0,C 180,E1 -26642.939,E2 -26642.939} C_VEL
LIN {X 0,Y 136.922,Z 341.637,A -85,B 0,C 180,E1 -26648.861,E2 -26648.861} C_VEL
LIN {X 0,Y 137.085,Z 343.66,A -85,B 0,C 180,E1 -26654.856,E2 -26654.856} C_VEL
LIN {X 0,Y 137.268,Z 345.267,A -85,B 0,C 180,E1 -26657.894,E2 -26657.894} C_VEL
LIN {X 0,Y 137.506,Z 347.219,A -85,B 0,C 180,E1 -26660.967,E2 -26660.967} C_VEL
LIN {X 0,Y 137.726,Z 351.188,A -85,B 0,C 180,E1 -26665.709,E2 -26665.709} C_VEL
LIN {X 0,Y 137.694,Z 356.357,A -85,B 0,C 180,E1 -26670.695,E2 -26670.695} C_VEL
LIN {X 0,Y 137.309,Z 361.446,A -85,B 0,C 180,E1 -26675.024,E2 -26675.024} C_VEL
LIN {X 0,Y 136.629,Z 364.278,A -85,B 0,C 180,E1 -26677.131,E2 -26677.131} C_VEL
LIN {X 0,Y 134.691,Z 368.319,A -85,B 0,C 180,E1 -26679.681,E2 -26679.681} C_VEL
LIN {X 0,Y 132.532,Z 372.018,A -85,B 0,C 180,E1 -26682.065,E2 -26682.065} C_VEL
LIN {X 0,Y 130.386,Z 374.331,A -85,B 0,C 180,E1 -26683.31,E2 -26683.31} C_VEL
LIN {X 0,Y 123.539,Z 380.392,A -85,B 0,C 180,E1 -26686.949,E2 -26686.949} C_VEL
LIN {X 0,Y 117.759,Z 385.016,A -85,B 0,C 180,E1 -26690.888,E2 -26690.888} C_VEL
LIN {X 0,Y 112.033,Z 388.956,A -85,B 0,C 180,E1 -26695.628,E2 -26695.628} C_VEL
LIN {X 0,Y 105.888,Z 392.442,A -85,B 0,C 180,E1 -26702.316,E2 -26702.316} C_VEL
LIN {X 0,Y 101.431,Z 394.266,A -85,B 0,C 180,E1 -26709.731,E2 -26709.731} C_VEL
LIN {X 0,Y 98.913,Z 394.584,A -85,B 0,C 180,E1 -26717.693,E2 -26717.693} C_VEL
LIN {X 0,Y 98.269,Z 394.154,A -85,B 0,C 180,E1 -26721.777,E2 -26721.777} C_VEL
LIN {X 0,Y 98.054,Z 393.311,A -85,B 0,C 180,E1 -26725.89,E2 -26725.89} C_VEL
LIN {X 0,Y 98.152,Z 392.075,A -85,B 0,C 180,E1 -26730,E2 -26730} C_VEL
LIN {X 0,Y 98.117,Z 389.376,A -85,B 0,C 180,E1 -26736.168,E2 -26736.168} C_VEL
LIN {X 0,Y 98.82,Z 385.629,A -85,B 0,C 180,E1 -26742.319,E2 -26742.319} C_VEL
LIN {X 0,Y 100.351,Z 380.728,A -85,B 0,C 180,E1 -26748.37,E2 -26748.37} C_VEL
LIN {X 0,Y 102.985,Z 374.544,A -85,B 0,C 180,E1 -26754.17,E2 -26754.17} C_VEL
LIN {X 0,Y 106.44,Z 366.817,A -85,B 0,C 180,E1 -26759.683,E2 -26759.683} C_VEL
LIN {X 0,Y 108.97,Z 360.892,A -85,B 0,C 180,E1 -26763.017,E2 -26763.017} C_VEL
LIN {X 0,Y 112.346,Z 353.283,A -85,B 0,C 180,E1 -26766.461,E2 -26766.461} C_VEL
LIN {X 0,Y 114.088,Z 344.278,A -85,B 0,C 180,E1 -26770.301,E2 -26770.301} C_VEL
LIN {X 0,Y 115.275,Z 334.774,A -85,B 0,C 180,E1 -26773.822,E2 -26773.822} C_VEL
LIN {X 0,Y 115.624,Z 324.058,A -85,B 0,C 180,E1 -26777.433,E2 -26777.433} C_VEL
LIN {X 0,Y 115.334,Z 320.98,A -85,B 0,C 180,E1 -26778.521,E2 -26778.521} C_VEL
LIN {X 0,Y 112.513,Z 311.96,A -85,B 0,C 180,E1 -26782.476,E2 -26782.476} C_VEL
LIN {X 0,Y 109.432,Z 304.67,A -85,B 0,C 180,E1 -26786.082,E2 -26786.082} C_VEL
LIN {X 0,Y 106.869,Z 300.561,A -85,B 0,C 180,E1 -26788.75,E2 -26788.75} C_VEL
LIN {X 0,Y 104.819,Z 297.571,A -85,B 0,C 180,E1 -26790.909,E2 -26790.909} C_VEL
LIN {X 0,Y 104.111,Z 296.123,A -85,B 0,C 180,E1 -26791.796,E2 -26791.796} C_VEL
LIN {X 0,Y 101.918,Z 294.085,A -85,B 0,C 180,E1 -26794.112,E2 -26794.112} C_VEL
LIN {X 0,Y 100.903,Z 291.547,A -85,B 0,C 180,E1 -26795.58,E2 -26795.58} C_VEL
LIN {X 0,Y 100.804,Z 290.919,A -85,B 0,C 180,E1 -26795.815,E2 -26795.815} C_VEL
LIN {X 0,Y 100.918,Z 290.91,A -85,B 0,C 180,E1 -26803.821,E2 -26803.821} C_VEL
LIN {X 0,Y 101.158,Z 290.876,A -85,B 0,C 180,E1 -26807.965,E2 -26807.965} C_VEL
LIN {X 0,Y 101.241,Z 290.877,A -85,B 0,C 180,E1 -26812.015,E2 -26812.015} C_VEL
LIN {X 0,Y 101.843,Z 290.749,A -85,B 0,C 180,E1 -26819.995,E2 -26819.995} C_VEL
LIN {X 0,Y 101.264,Z 290.866,A -85,B 0,C 180,E1 -26827.974,E2 -26827.974} C_VEL
LIN {X 0,Y 101.121,Z 290.89,A -85,B 0,C 180,E1 -26833.346,E2 -26833.346} C_VEL
LIN {X 0,Y 100.811,Z 290.927,A -85,B 0,C 180,E1 -26840.395,E2 -26840.395} C_VEL
LIN {X 0,Y 100.77,Z 290.921,A -85,B 0,C 180,E1 -26844.954,E2 -26844.954} C_VEL
LIN {X 0,Y 100.699,Z 290.938,A -85,B 0,C 180,E1 -26853.124,E2 -26853.124} C_VEL
LIN {X 0,Y 100.696,Z 291.005,A -85,B 0,C 180,E1 -26857.791,E2 -26857.791} C_VEL
LIN {X 0,Y 101.588,Z 293.601,A -85,B 0,C 180,E1 -26859.283,E2 -26859.283} C_VEL
LIN {X 0,Y 103.598,Z 295.788,A -85,B 0,C 180,E1 -26861.553,E2 -26861.553} C_VEL
LIN {X 0,Y 104.257,Z 296.615,A -85,B 0,C 180,E1 -26862.277,E2 -26862.277} C_VEL
LIN {X 0,Y 104.943,Z 298.218,A -85,B 0,C 180,E1 -26863.234,E2 -26863.234} C_VEL
LIN {X 0,Y 106.583,Z 302.168,A -85,B 0,C 180,E1 -26865.458,E2 -26865.458} C_VEL
LIN {X 0,Y 107.632,Z 306.697,A -85,B 0,C 180,E1 -26867.456,E2 -26867.456} C_VEL
LIN {X 0,Y 109.359,Z 319.312,A -85,B 0,C 180,E1 -26872.627,E2 -26872.627} C_VEL
LIN {X 0,Y 110.106,Z 322.158,A -85,B 0,C 180,E1 -26874.052,E2 -26874.052} C_VEL
LIN {X 0,Y 110.778,Z 325.208,A -85,B 0,C 180,E1 -26875.554,E2 -26875.554} C_VEL
LIN {X 0,Y 110.793,Z 333.518,A -85,B 0,C 180,E1 -26879.008,E2 -26879.008} C_VEL
LIN {X 0,Y 109.928,Z 341.429,A -85,B 0,C 180,E1 -26882.386,E2 -26882.386} C_VEL
LIN {X 0,Y 106.316,Z 349.652,A -85,B 0,C 180,E1 -26885.597,E2 -26885.597} C_VEL
LIN {X 0,Y 102.241,Z 358.216,A -85,B 0,C 180,E1 -26889.898,E2 -26889.898} C_VEL
LIN {X 0,Y 98.106,Z 366.542,A -85,B 0,C 180,E1 -26895.48,E2 -26895.48} C_VEL
LIN {X 0,Y 94.951,Z 373.246,A -85,B 0,C 180,E1 -26901.487,E2 -26901.487} C_VEL
LIN {X 0,Y 92.687,Z 378.604,A -85,B 0,C 180,E1 -26907.827,E2 -26907.827} C_VEL
LIN {X 0,Y 91.24,Z 382.799,A -85,B 0,C 180,E1 -26914.417,E2 -26914.417} C_VEL
LIN {X 0,Y 90.667,Z 385.02,A -85,B 0,C 180,E1 -26918.918,E2 -26918.918} C_VEL
LIN {X 0,Y 90.486,Z 386.761,A -85,B 0,C 180,E1 -26923.474,E2 -26923.474} C_VEL
LIN {X 0,Y 90.821,Z 388.088,A -85,B 0,C 180,E1 -26928.03,E2 -26928.03} C_VEL
LIN {X 0,Y 91.651,Z 389.085,A -85,B 0,C 180,E1 -26933.062,E2 -26933.062} C_VEL
LIN {X 0,Y 94.334,Z 389.556,A -85,B 0,C 180,E1 -26941.432,E2 -26941.432} C_VEL
LIN {X 0,Y 97.829,Z 388.853,A -85,B 0,C 180,E1 -26947.801,E2 -26947.801} C_VEL
LIN {X 0,Y 102.093,Z 387.241,A -85,B 0,C 180,E1 -26953.502,E2 -26953.502} C_VEL
LIN {X 0,Y 108.298,Z 384.115,A -85,B 0,C 180,E1 -26959.544,E2 -26959.544} C_VEL
LIN {X 0,Y 115.745,Z 379.414,A -85,B 0,C 180,E1 -26965.054,E2 -26965.054} C_VEL
LIN {X 0,Y 124.007,Z 373.036,A -85,B 0,C 180,E1 -26969.798,E2 -26969.798} C_VEL
LIN {X 0,Y 129.056,Z 368.562,A -85,B 0,C 180,E1 -26972.24,E2 -26972.24} C_VEL
LIN {X 0,Y 130.225,Z 367.283,A -85,B 0,C 180,E1 -26972.93,E2 -26972.93} C_VEL
LIN {X 0,Y 131.574,Z 364.474,A -85,B 0,C 180,E1 -26975.234,E2 -26975.234} C_VEL
LIN {X 0,Y 132.361,Z 361.369,A -85,B 0,C 180,E1 -26978.185,E2 -26978.185} C_VEL
LIN {X 0,Y 132.874,Z 357.553,A -85,B 0,C 180,E1 -26982.182,E2 -26982.182} C_VEL
LIN {X 0,Y 133.11,Z 354.098,A -85,B 0,C 180,E1 -26986.259,E2 -26986.259} C_VEL
LIN {X 0,Y 133.13,Z 350.916,A -85,B 0,C 180,E1 -26990.891,E2 -26990.891} C_VEL
LIN {X 0,Y 133.106,Z 349.196,A -85,B 0,C 180,E1 -26993.942,E2 -26993.942} C_VEL
LIN {X 0,Y 133.095,Z 347.875,A -85,B 0,C 180,E1 -26996.977,E2 -26996.977} C_VEL
LIN {X 0,Y 132.99,Z 346.995,A -85,B 0,C 180,E1 -27000.004,E2 -27000.004} C_VEL
LIN {X 0,Y 132.843,Z 346.602,A -85,B 0,C 180,E1 -27003.036,E2 -27003.036} C_VEL
LIN {X 0,Y 132.594,Z 346.791,A -85,B 0,C 180,E1 -27006.089,E2 -27006.089} C_VEL
LIN {X 0,Y 132.488,Z 347.312,A -85,B 0,C 180,E1 -27009.161,E2 -27009.161} C_VEL
LIN {X 0,Y 132.459,Z 348.21,A -85,B 0,C 180,E1 -27012.257,E2 -27012.257} C_VEL
LIN {X 0,Y 132.564,Z 350.423,A -85,B 0,C 180,E1 -27017.396,E2 -27017.396} C_VEL
LIN {X 0,Y 132.572,Z 353.277,A -85,B 0,C 180,E1 -27021.786,E2 -27021.786} C_VEL
LIN {X 0,Y 132.496,Z 356.3,A -85,B 0,C 180,E1 -27025.617,E2 -27025.617} C_VEL
LIN {X 0,Y 132.145,Z 360.439,A -85,B 0,C 180,E1 -27029.954,E2 -27029.954} C_VEL
LIN {X 0,Y 131.489,Z 364.826,A -85,B 0,C 180,E1 -27034.074,E2 -27034.074} C_VEL
LIN {X 0,Y 130.436,Z 367.707,A -85,B 0,C 180,E1 -27036.352,E2 -27036.352} C_VEL
LIN {X 0,Y 126.769,Z 373.5,A -85,B 0,C 180,E1 -27040.335,E2 -27040.335} C_VEL
LIN {X 0,Y 118.454,Z 380.577,A -85,B 0,C 180,E1 -27044.606,E2 -27044.606} C_VEL
LIN {X 0,Y 111.842,Z 385.459,A -85,B 0,C 180,E1 -27048.95,E2 -27048.95} C_VEL
LIN {X 0,Y 106.25,Z 388.982,A -85,B 0,C 180,E1 -27053.466,E2 -27053.466} C_VEL
LIN {X 0,Y 102.717,Z 390.891,A -85,B 0,C 180,E1 -27056.814,E2 -27056.814} C_VEL
LIN {X 0,Y 99.645,Z 392.372,A -85,B 0,C 180,E1 -27060.416,E2 -27060.416} C_VEL
LIN {X 0,Y 94.767,Z 394.116,A -85,B 0,C 180,E1 -27068.236,E2 -27068.236} C_VEL
LIN {X 0,Y 91.958,Z 394.359,A -85,B 0,C 180,E1 -27076.746,E2 -27076.746} C_VEL
LIN {X 0,Y 90.982,Z 392.995,A -85,B 0,C 180,E1 -27085.57,E2 -27085.57} C_VEL
LIN {X 0,Y 91.056,Z 391.726,A -85,B 0,C 180,E1 -27090,E2 -27090} C_VEL
LIN {X 0,Y 91.067,Z 388.958,A -85,B 0,C 180,E1 -27096.648,E2 -27096.648} C_VEL
LIN {X 0,Y 91.86,Z 385.134,A -85,B 0,C 180,E1 -27103.269,E2 -27103.269} C_VEL
LIN {X 0,Y 93.596,Z 380.152,A -85,B 0,C 180,E1 -27109.749,E2 -27109.749} C_VEL
LIN {X 0,Y 96.509,Z 373.88,A -85,B 0,C 180,E1 -27115.908,E2 -27115.908} C_VEL
LIN {X 0,Y 100.245,Z 365.996,A -85,B 0,C 180,E1 -27121.722,E2 -27121.722} C_VEL
LIN {X 0,Y 103.258,Z 359.654,A -85,B 0,C 180,E1 -27125.365,E2 -27125.365} C_VEL
LIN {X 0,Y 106.152,Z 353.239,A -85,B 0,C 180,E1 -27128.366,E2 -27128.366} C_VEL
LIN {X 0,Y 108.237,Z 343.394,A -85,B 0,C 180,E1 -27132.774,E2 -27132.774} C_VEL
LIN {X 0,Y 109.469,Z 334.057,A -85,B 0,C 180,E1 -27136.427,E2 -27136.427} C_VEL
LIN {X 0,Y 109.938,Z 325.178,A -85,B 0,C 180,E1 -27139.625,E2 -27139.625} C_VEL
LIN {X 0,Y 107.858,Z 317.197,A -85,B 0,C 180,E1 -27143.454,E2 -27143.454} C_VEL
LIN {X 0,Y 105.668,Z 311.069,A -85,B 0,C 180,E1 -27146.717,E2 -27146.717} C_VEL
LIN {X 0,Y 103.581,Z 306.867,A -85,B 0,C 180,E1 -27149.406,E2 -27149.406} C_VEL
LIN {X 0,Y 100.987,Z 302.632,A -85,B 0,C 180,E1 -27152.68,E2 -27152.68} C_VEL
LIN {X 0,Y 98.38,Z 299.251,A -85,B 0,C 180,E1 -27156.086,E2 -27156.086} C_VEL
LIN {X 0,Y 97.533,Z 297.177,A -85,B 0,C 180,E1 -27157.551,E2 -27157.551} C_VEL
LIN {X 0,Y 95.164,Z 295.22,A -85,B 0,C 180,E1 -27160.865,E2 -27160.865} C_VEL
LIN {X 0,Y 94.042,Z 292.914,A -85,B 0,C 180,E1 -27163.058,E2 -27163.058} C_VEL
LIN {X 0,Y 93.873,Z 291.787,A -85,B 0,C 180,E1 -27163.786,E2 -27163.786} C_VEL
LIN {X 0,Y 94.068,Z 291.764,A -85,B 0,C 180,E1 -27167.043,E2 -27167.043} C_VEL
LIN {X 0,Y 94.175,Z 291.755,A -85,B 0,C 180,E1 -27171.411,E2 -27171.411} C_VEL
LIN {X 0,Y 94.772,Z 291.629,A -85,B 0,C 180,E1 -27179.995,E2 -27179.995} C_VEL
LIN {X 0,Y 94.197,Z 291.742,A -85,B 0,C 180,E1 -27188.576,E2 -27188.576} C_VEL
LIN {X 0,Y 94.039,Z 291.771,A -85,B 0,C 180,E1 -27193.703,E2 -27193.703} C_VEL
LIN {X 0,Y 93.688,Z 291.806,A -85,B 0,C 180,E1 -27202.023,E2 -27202.023} C_VEL
LIN {X 0,Y 93.617,Z 291.821,A -85,B 0,C 180,E1 -27206.765,E2 -27206.765} C_VEL
LIN {X 0,Y 93.593,Z 291.832,A -85,B 0,C 180,E1 -27209.672,E2 -27209.672} C_VEL
LIN {X 0,Y 94.394,Z 294.314,A -85,B 0,C 180,E1 -27211.685,E2 -27211.685} C_VEL
LIN {X 0,Y 96.851,Z 296.91,A -85,B 0,C 180,E1 -27215.481,E2 -27215.481} C_VEL
LIN {X 0,Y 97.578,Z 297.508,A -85,B 0,C 180,E1 -27216.451,E2 -27216.451} C_VEL
LIN {X 0,Y 99.158,Z 300.717,A -85,B 0,C 180,E1 -27219.097,E2 -27219.097} C_VEL
LIN {X 0,Y 100.429,Z 301.951,A -85,B 0,C 180,E1 -27220.631,E2 -27220.631} C_VEL
LIN {X 0,Y 102.317,Z 305.54,A -85,B 0,C 180,E1 -27223.377,E2 -27223.377} C_VEL
LIN {X 0,Y 103.122,Z 306.529,A -85,B 0,C 180,E1 -27224.305,E2 -27224.305} C_VEL
LIN {X 0,Y 107.747,Z 315.967,A -85,B 0,C 180,E1 -27230.546,E2 -27230.546} C_VEL
LIN {X 0,Y 110.106,Z 322.158,A -85,B 0,C 180,E1 -27234.052,E2 -27234.052} C_VEL
LIN {X 0,Y 110.556,Z 325.075,A -85,B 0,C 180,E1 -27235.378,E2 -27235.378} C_VEL
LIN {X 0,Y 109.818,Z 329.989,A -85,B 0,C 180,E1 -27237.046,E2 -27237.046} C_VEL
LIN {X 0,Y 107.934,Z 335.009,A -85,B 0,C 180,E1 -27238.467,E2 -27238.467} C_VEL
LIN {X 0,Y 102.653,Z 345.022,A -85,B 0,C 180,E1 -27241.46,E2 -27241.46} C_VEL
LIN {X 0,Y 101.103,Z 348.153,A -85,B 0,C 180,E1 -27242.732,E2 -27242.732} C_VEL
LIN {X 0,Y 96.392,Z 357.611,A -85,B 0,C 180,E1 -27247.494,E2 -27247.494} C_VEL
LIN {X 0,Y 92.613,Z 364.827,A -85,B 0,C 180,E1 -27252.33,E2 -27252.33} C_VEL
LIN {X 0,Y 88.865,Z 371.921,A -85,B 0,C 180,E1 -27258.597,E2 -27258.597} C_VEL
LIN {X 0,Y 86.178,Z 377.579,A -85,B 0,C 180,E1 -27265.322,E2 -27265.322} C_VEL
LIN {X 0,Y 84.425,Z 382.239,A -85,B 0,C 180,E1 -27272.758,E2 -27272.758} C_VEL
LIN {X 0,Y 83.502,Z 385.449,A -85,B 0,C 180,E1 -27279.69,E2 -27279.69} C_VEL
LIN {X 0,Y 83.416,Z 387.149,A -85,B 0,C 180,E1 -27284.64,E2 -27284.64} C_VEL
LIN {X 0,Y 83.88,Z 388.437,A -85,B 0,C 180,E1 -27289.581,E2 -27289.581} C_VEL
LIN {X 0,Y 84.789,Z 389.297,A -85,B 0,C 180,E1 -27294.483,E2 -27294.483} C_VEL
LIN {X 0,Y 86.194,Z 389.719,A -85,B 0,C 180,E1 -27299.288,E2 -27299.288} C_VEL
LIN {X 0,Y 88.116,Z 389.743,A -85,B 0,C 180,E1 -27303.938,E2 -27303.938} C_VEL
LIN {X 0,Y 91.605,Z 389.092,A -85,B 0,C 180,E1 -27309.905,E2 -27309.905} C_VEL
LIN {X 0,Y 96.848,Z 387.263,A -85,B 0,C 180,E1 -27316.523,E2 -27316.523} C_VEL
LIN {X 0,Y 102.949,Z 384.41,A -85,B 0,C 180,E1 -27322.098,E2 -27322.098} C_VEL
LIN {X 0,Y 109.315,Z 380.728,A -85,B 0,C 180,E1 -27326.696,E2 -27326.696} C_VEL
LIN {X 0,Y 117.674,Z 374.944,A -85,B 0,C 180,E1 -27331.463,E2 -27331.463} C_VEL
LIN {X 0,Y 124.424,Z 369.366,A -85,B 0,C 180,E1 -27334.652,E2 -27334.652} C_VEL
LIN {X 0,Y 125.861,Z 366.78,A -85,B 0,C 180,E1 -27336.995,E2 -27336.995} C_VEL
LIN {X 0,Y 126.881,Z 363.467,A -85,B 0,C 180,E1 -27340.593,E2 -27340.593} C_VEL
LIN {X 0,Y 127.657,Z 359.384,A -85,B 0,C 180,E1 -27345.66,E2 -27345.66} C_VEL
LIN {X 0,Y 128.021,Z 355.839,A -85,B 0,C 180,E1 -27351.16,E2 -27351.16} C_VEL
LIN {X 0,Y 128.22,Z 353.174,A -85,B 0,C 180,E1 -27356.862,E2 -27356.862} C_VEL
LIN {X 0,Y 128.251,Z 352.312,A -85,B 0,C 180,E1 -27360.004,E2 -27360.004} C_VEL
LIN {X 0,Y 128.147,Z 351.945,A -85,B 0,C 180,E1 -27363.148,E2 -27363.148} C_VEL
LIN {X 0,Y 127.787,Z 352.467,A -85,B 0,C 180,E1 -27368.138,E2 -27368.138} C_VEL
LIN {X 0,Y 127.614,Z 353.693,A -85,B 0,C 180,E1 -27372.73,E2 -27372.73} C_VEL
LIN {X 0,Y 127.595,Z 354.942,A -85,B 0,C 180,E1 -27375.99,E2 -27375.99} C_VEL
LIN {X 0,Y 127.444,Z 357.386,A -85,B 0,C 180,E1 -27380.372,E2 -27380.372} C_VEL
LIN {X 0,Y 127.141,Z 360.272,A -85,B 0,C 180,E1 -27384.497,E2 -27384.497} C_VEL
LIN {X 0,Y 126.623,Z 363.367,A -85,B 0,C 180,E1 -27388.152,E2 -27388.152} C_VEL
LIN {X 0,Y 125.604,Z 367.904,A -85,B 0,C 180,E1 -27392.936,E2 -27392.936} C_VEL
LIN {X 0,Y 124.552,Z 370.226,A -85,B 0,C 180,E1 -27394.956,E2 -27394.956} C_VEL
LIN {X 0,Y 121.065,Z 374.882,A -85,B 0,C 180,E1 -27398.402,E2 -27398.402} C_VEL
LIN {X 0,Y 113.578,Z 380.762,A -85,B 0,C 180,E1 -27402.053,E2 -27402.053} C_VEL
LIN {X 0,Y 106.034,Z 385.909,A -85,B 0,C 180,E1 -27406.816,E2 -27406.816} C_VEL
LIN {X 0,Y 100.634,Z 389.009,A -85,B 0,C 180,E1 -27411.059,E2 -27411.059} C_VEL
LIN {X 0,Y 96.838,Z 390.875,A -85,B 0,C 180,E1 -27414.509,E2 -27414.509} C_VEL
LIN {X 0,Y 90.598,Z 393.317,A -85,B 0,C 180,E1 -27422.262,E2 -27422.262} C_VEL
LIN {X 0,Y 86.362,Z 394.244,A -85,B 0,C 180,E1 -27431.004,E2 -27431.004} C_VEL
LIN {X 0,Y 85.041,Z 394.113,A -85,B 0,C 180,E1 -27435.646,E2 -27435.646} C_VEL
LIN {X 0,Y 83.901,Z 392.675,A -85,B 0,C 180,E1 -27445.195,E2 -27445.195} C_VEL
LIN {X 0,Y 83.954,Z 391.371,A -85,B 0,C 180,E1 -27450,E2 -27450} C_VEL
LIN {X 0,Y 84,Z 388.53,A -85,B 0,C 180,E1 -27457.21,E2 -27457.21} C_VEL
LIN {X 0,Y 84.94,Z 384.629,A -85,B 0,C 180,E1 -27464.372,E2 -27464.372} C_VEL
LIN {X 0,Y 86.912,Z 379.564,A -85,B 0,C 180,E1 -27471.339,E2 -27471.339} C_VEL
LIN {X 0,Y 90.142,Z 373.19,A -85,B 0,C 180,E1 -27477.891,E2 -27477.891} C_VEL
LIN {X 0,Y 94.177,Z 365.148,A -85,B 0,C 180,E1 -27484.034,E2 -27484.034} C_VEL
LIN {X 0,Y 97.516,Z 358.766,A -85,B 0,C 180,E1 -27487.774,E2 -27487.774} C_VEL
LIN {X 0,Y 99.345,Z 355.161,A -85,B 0,C 180,E1 -27489.544,E2 -27489.544} C_VEL
LIN {X 0,Y 101.417,Z 347.764,A -85,B 0,C 180,E1 -27493.181,E2 -27493.181} C_VEL
LIN {X 0,Y 103.141,Z 338.98,A -85,B 0,C 180,E1 -27497.041,E2 -27497.041} C_VEL
LIN {X 0,Y 104.291,Z 328.496,A -85,B 0,C 180,E1 -27501.216,E2 -27501.216} C_VEL
LIN {X 0,Y 103.011,Z 322.095,A -85,B 0,C 180,E1 -27504.552,E2 -27504.552} C_VEL
LIN {X 0,Y 100.928,Z 315.312,A -85,B 0,C 180,E1 -27508.511,E2 -27508.511} C_VEL
LIN {X 0,Y 98.375,Z 310.46,A -85,B 0,C 180,E1 -27512.326,E2 -27512.326} C_VEL
LIN {X 0,Y 97.178,Z 308.018,A -85,B 0,C 180,E1 -27514.278,E2 -27514.278} C_VEL
LIN {X 0,Y 95.263,Z 305.41,A -85,B 0,C 180,E1 -27517.207,E2 -27517.207} C_VEL
LIN {X 0,Y 94.337,Z 303.364,A -85,B 0,C 180,E1 -27518.985,E2 -27518.985} C_VEL
LIN {X 0,Y 92.042,Z 300.829,A -85,B 0,C 180,E1 -27522.927,E2 -27522.927} C_VEL
LIN {X 0,Y 91.067,Z 298.264,A -85,B 0,C 180,E1 -27525.503,E2 -27525.503} C_VEL
LIN {X 0,Y 88.206,Z 295.622,A -85,B 0,C 180,E1 -27532.555,E2 -27532.555} C_VEL
LIN {X 0,Y 87.414,Z 293.263,A -85,B 0,C 180,E1 -27536.682,E2 -27536.682} C_VEL
LIN {X 0,Y 87.398,Z 292.549,A -85,B 0,C 180,E1 -27537.69,E2 -27537.69} C_VEL
LIN {X 0,Y 87.701,Z 292.508,A -85,B 0,C 180,E1 -27539.995,E2 -27539.995} C_VEL
LIN {X 0,Y 87.105,Z 292.622,A -85,B 0,C 180,E1 -27549.281,E2 -27549.281} C_VEL
LIN {X 0,Y 86.927,Z 292.8,A -85,B 0,C 180,E1 -27554.568,E2 -27554.568} C_VEL
LIN {X 0,Y 87.765,Z 295.757,A -85,B 0,C 180,E1 -27560.196,E2 -27560.196} C_VEL
LIN {X 0,Y 90.966,Z 298.591,A -85,B 0,C 180,E1 -27568.394,E2 -27568.394} C_VEL
LIN {X 0,Y 92.221,Z 301.441,A -85,B 0,C 180,E1 -27571.59,E2 -27571.59} C_VEL
LIN {X 0,Y 94.089,Z 303.337,A -85,B 0,C 180,E1 -27574.752,E2 -27574.752} C_VEL
LIN {X 0,Y 95.903,Z 306.828,A -85,B 0,C 180,E1 -27578.18,E2 -27578.18} C_VEL
LIN {X 0,Y 96.737,Z 307.747,A -85,B 0,C 180,E1 -27579.359,E2 -27579.359} C_VEL
LIN {X 0,Y 99.953,Z 314.04,A -85,B 0,C 180,E1 -27584.671,E2 -27584.671} C_VEL
LIN {X 0,Y 103.01,Z 321.077,A -85,B 0,C 180,E1 -27589.689,E2 -27589.689} C_VEL
LIN {X 0,Y 104.991,Z 327.148,A -85,B 0,C 180,E1 -27593.435,E2 -27593.435} C_VEL
LIN {X 0,Y 104.833,Z 335.021,A -85,B 0,C 180,E1 -27597.054,E2 -27597.054} C_VEL
LIN {X 0,Y 104.082,Z 341.631,A -85,B 0,C 180,E1 -27600.134,E2 -27600.134} C_VEL
LIN {X 0,Y 101.103,Z 348.153,A -85,B 0,C 180,E1 -27602.732,E2 -27602.732} C_VEL
LIN {X 0,Y 98.549,Z 352.463,A -85,B 0,C 180,E1 -27604.539,E2 -27604.539} C_VEL
LIN {X 0,Y 92.694,Z 359.065,A -85,B 0,C 180,E1 -27607.267,E2 -27607.267} C_VEL
LIN {X 0,Y 86.742,Z 365.101,A -85,B 0,C 180,E1 -27610.612,E2 -27610.612} C_VEL
LIN {X 0,Y 84.168,Z 368.507,A -85,B 0,C 180,E1 -27613.373,E2 -27613.373} C_VEL
LIN {X 0,Y 80.871,Z 374.635,A -85,B 0,C 180,E1 -27619.991,E2 -27619.991} C_VEL
LIN {X 0,Y 78.415,Z 379.78,A -85,B 0,C 180,E1 -27627.431,E2 -27627.431} C_VEL
LIN {X 0,Y 76.86,Z 383.799,A -85,B 0,C 180,E1 -27635.246,E2 -27635.246} C_VEL
LIN {X 0,Y 76.344,Z 385.879,A -85,B 0,C 180,E1 -27640.609,E2 -27640.609} C_VEL
LIN {X 0,Y 76.377,Z 387.538,A -85,B 0,C 180,E1 -27646.024,E2 -27646.024} C_VEL
LIN {X 0,Y 77.819,Z 389.427,A -85,B 0,C 180,E1 -27655.444,E2 -27655.444} C_VEL
LIN {X 0,Y 79.845,Z 389.946,A -85,B 0,C 180,E1 -27661.877,E2 -27661.877} C_VEL
LIN {X 0,Y 82.108,Z 389.929,A -85,B 0,C 180,E1 -27666.808,E2 -27666.808} C_VEL
LIN {X 0,Y 85.48,Z 389.339,A -85,B 0,C 180,E1 -27672.281,E2 -27672.281} C_VEL
LIN {X 0,Y 91.903,Z 387.284,A -85,B 0,C 180,E1 -27679.88,E2 -27679.88} C_VEL
LIN {X 0,Y 97.78,Z 384.722,A -85,B 0,C 180,E1 -27684.906,E2 -27684.906} C_VEL
LIN {X 0,Y 105.435,Z 380.571,A -85,B 0,C 180,E1 -27690.057,E2 -27690.057} C_VEL
LIN {X 0,Y 113.443,Z 375.298,A -85,B 0,C 180,E1 -27694.305,E2 -27694.305} C_VEL
LIN {X 0,Y 118.631,Z 371.288,A -85,B 0,C 180,E1 -27696.67,E2 -27696.67} C_VEL
LIN {X 0,Y 119.52,Z 370.258,A -85,B 0,C 180,E1 -27697.536,E2 -27697.536} C_VEL
LIN {X 0,Y 120.701,Z 367.699,A -85,B 0,C 180,E1 -27700.538,E2 -27700.538} C_VEL
LIN {X 0,Y 121.762,Z 364.389,A -85,B 0,C 180,E1 -27704.95,E2 -27704.95} C_VEL
LIN {X 0,Y 122.494,Z 361.189,A -85,B 0,C 180,E1 -27710.093,E2 -27710.093} C_VEL
LIN {X 0,Y 122.812,Z 359.547,A -85,B 0,C 180,E1 -27713.432,E2 -27713.432} C_VEL
LIN {X 0,Y 123.037,Z 358.221,A -85,B 0,C 180,E1 -27716.729,E2 -27716.729} C_VEL
LIN {X 0,Y 123.193,Z 357.332,A -85,B 0,C 180,E1 -27720.004,E2 -27720.004} C_VEL
LIN {X 0,Y 123.141,Z 357.005,A -85,B 0,C 180,E1 -27723.276,E2 -27723.276} C_VEL
LIN {X 0,Y 122.875,Z 357.261,A -85,B 0,C 180,E1 -27726.572,E2 -27726.572} C_VEL
LIN {X 0,Y 122.498,Z 358.692,A -85,B 0,C 180,E1 -27732.76,E2 -27732.76} C_VEL
LIN {X 0,Y 122.296,Z 360.25,A -85,B 0,C 180,E1 -27736.702,E2 -27736.702} C_VEL
LIN {X 0,Y 122.001,Z 362.112,A -85,B 0,C 180,E1 -27740.225,E2 -27740.225} C_VEL
LIN {X 0,Y 121.552,Z 364.464,A -85,B 0,C 180,E1 -27743.878,E2 -27743.878} C_VEL
LIN {X 0,Y 120.44,Z 368.436,A -85,B 0,C 180,E1 -27748.924,E2 -27748.924} C_VEL
LIN {X 0,Y 119.568,Z 371.029,A -85,B 0,C 180,E1 -27751.943,E2 -27751.943} C_VEL
LIN {X 0,Y 118.349,Z 373.013,A -85,B 0,C 180,E1 -27753.763,E2 -27753.763} C_VEL
LIN {X 0,Y 116.556,Z 375.173,A -85,B 0,C 180,E1 -27755.513,E2 -27755.513} C_VEL
LIN {X 0,Y 115.488,Z 376.203,A -85,B 0,C 180,E1 -27756.264,E2 -27756.264} C_VEL
LIN {X 0,Y 106.478,Z 382.573,A -85,B 0,C 180,E1 -27760.622,E2 -27760.622} C_VEL
LIN {X 0,Y 99.506,Z 386.785,A -85,B 0,C 180,E1 -27765.068,E2 -27765.068} C_VEL
LIN {X 0,Y 95.201,Z 389.035,A -85,B 0,C 180,E1 -27768.365,E2 -27768.365} C_VEL
LIN {X 0,Y 91.14,Z 390.837,A -85,B 0,C 180,E1 -27771.912,E2 -27771.912} C_VEL
LIN {X 0,Y 84.375,Z 393.202,A -85,B 0,C 180,E1 -27780.016,E2 -27780.016} C_VEL
LIN {X 0,Y 81.688,Z 393.817,A -85,B 0,C 180,E1 -27784.522,E2 -27784.522} C_VEL
LIN {X 0,Y 79.659,Z 394.046,A -85,B 0,C 180,E1 -27789.336,E2 -27789.336} C_VEL
LIN {X 0,Y 77.215,Z 393.299,A -85,B 0,C 180,E1 -27799.512,E2 -27799.512} C_VEL
LIN {X 0,Y 76.843,Z 392.356,A -85,B 0,C 180,E1 -27804.753,E2 -27804.753} C_VEL
LIN {X 0,Y 76.86,Z 391.013,A -85,B 0,C 180,E1 -27810,E2 -27810} C_VEL
LIN {X 0,Y 76.958,Z 388.103,A -85,B 0,C 180,E1 -27817.873,E2 -27817.873} C_VEL
LIN {X 0,Y 78.037,Z 384.122,A -85,B 0,C 180,E1 -27825.675,E2 -27825.675} C_VEL
LIN {X 0,Y 80.795,Z 377.959,A -85,B 0,C 180,E1 -27834.404,E2 -27834.404} C_VEL
LIN {X 0,Y 84.576,Z 371.218,A -85,B 0,C 180,E1 -27841.288,E2 -27841.288} C_VEL
LIN {X 0,Y 88.104,Z 364.661,A -85,B 0,C 180,E1 -27846.408,E2 -27846.408} C_VEL
LIN {X 0,Y 92.969,Z 356.004,A -85,B 0,C 180,E1 -27851.409,E2 -27851.409} C_VEL
LIN {X 0,Y 95.048,Z 349.963,A -85,B 0,C 180,E1 -27854.622,E2 -27854.622} C_VEL
LIN {X 0,Y 97.239,Z 340.853,A -85,B 0,C 180,E1 -27858.998,E2 -27858.998} C_VEL
LIN {X 0,Y 98.684,Z 331.443,A -85,B 0,C 180,E1 -27863.092,E2 -27863.092} C_VEL
LIN {X 0,Y 97.871,Z 326.036,A -85,B 0,C 180,E1 -27866.179,E2 -27866.179} C_VEL
LIN {X 0,Y 96.126,Z 319.568,A -85,B 0,C 180,E1 -27870.424,E2 -27870.424} C_VEL
LIN {X 0,Y 93.432,Z 313.683,A -85,B 0,C 180,E1 -27875.556,E2 -27875.556} C_VEL
LIN {X 0,Y 91.736,Z 311.079,A -85,B 0,C 180,E1 -27878.655,E2 -27878.655} C_VEL
LIN {X 0,Y 91.305,Z 309.923,A -85,B 0,C 180,E1 -27879.729,E2 -27879.729} C_VEL
LIN {X 0,Y 89.209,Z 307.134,A -85,B 0,C 180,E1 -27883.989,E2 -27883.989} C_VEL
LIN {X 0,Y 88.534,Z 305.191,A -85,B 0,C 180,E1 -27886.217,E2 -27886.217} C_VEL
LIN {X 0,Y 85.588,Z 300.939,A -85,B 0,C 180,E1 -27896.169,E2 -27896.169} C_VEL
LIN {X 0,Y 85.415,Z 299.311,A -85,B 0,C 180,E1 -27898.816,E2 -27898.816} C_VEL
LIN {X 0,Y 85.022,Z 299.502,A -85,B 0,C 180,E1 -27913.348,E2 -27913.348} C_VEL
LIN {X 0,Y 85.58,Z 302.328,A -85,B 0,C 180,E1 -27919.171,E2 -27919.171} C_VEL
LIN {X 0,Y 87.739,Z 304.626,A -85,B 0,C 180,E1 -27926.133,E2 -27926.133} C_VEL
LIN {X 0,Y 89.351,Z 307.784,A -85,B 0,C 180,E1 -27930.739,E2 -27930.739} C_VEL
LIN {X 0,Y 90.439,Z 309.014,A -85,B 0,C 180,E1 -27932.947,E2 -27932.947} C_VEL
LIN {X 0,Y 93.09,Z 313.848,A -85,B 0,C 180,E1 -27938.517,E2 -27938.517} C_VEL
LIN {X 0,Y 95.849,Z 320.034,A -85,B 0,C 180,E1 -27944.142,E2 -27944.142} C_VEL
LIN {X 0,Y 98.099,Z 326.019,A -85,B 0,C 180,E1 -27948.78,E2 -27948.78} C_VEL
LIN {X 0,Y 99.423,Z 331.062,A -85,B 0,C 180,E1 -27952.18,E2 -27952.18} C_VEL
LIN {X 0,Y 98.574,Z 339.7,A -85,B 0,C 180,E1 -27956.458,E2 -27956.458} C_VEL
LIN {X 0,Y 98.04,Z 342.886,A -85,B 0,C 180,E1 -27958.085,E2 -27958.085} C_VEL
LIN {X 0,Y 93.579,Z 351.842,A -85,B 0,C 180,E1 -27962.006,E2 -27962.006} C_VEL
LIN {X 0,Y 89.047,Z 360.079,A -85,B 0,C 180,E1 -27966.758,E2 -27966.758} C_VEL
LIN {X 0,Y 84.168,Z 368.507,A -85,B 0,C 180,E1 -27973.373,E2 -27973.373} C_VEL
LIN {X 0,Y 81.806,Z 371.706,A -85,B 0,C 180,E1 -27976.398,E2 -27976.398} C_VEL
LIN {X 0,Y 76.698,Z 376.46,A -85,B 0,C 180,E1 -27981.487,E2 -27981.487} C_VEL
LIN {X 0,Y 71.95,Z 380.507,A -85,B 0,C 180,E1 -27987.479,E2 -27987.479} C_VEL
LIN {X 0,Y 70.293,Z 382.581,A -85,B 0,C 180,E1 -27991.768,E2 -27991.768} C_VEL
LIN {X 0,Y 69.21,Z 386.308,A -85,B 0,C 180,E1 -28001.717,E2 -28001.717} C_VEL
LIN {X 0,Y 69.396,Z 387.927,A -85,B 0,C 180,E1 -28007.687,E2 -28007.687} C_VEL
LIN {X 0,Y 71.012,Z 389.6,A -85,B 0,C 180,E1 -28017.052,E2 -28017.052} C_VEL
LIN {X 0,Y 73.678,Z 390.174,A -85,B 0,C 180,E1 -28024.912,E2 -28024.912} C_VEL
LIN {X 0,Y 76.322,Z 390.112,A -85,B 0,C 180,E1 -28030.133,E2 -28030.133} C_VEL
LIN {X 0,Y 79.505,Z 389.589,A -85,B 0,C 180,E1 -28035.004,E2 -28035.004} C_VEL
LIN {X 0,Y 83.179,Z 388.654,A -85,B 0,C 180,E1 -28039.5,E2 -28039.5} C_VEL
LIN {X 0,Y 87.315,Z 387.306,A -85,B 0,C 180,E1 -28043.599,E2 -28043.599} C_VEL
LIN {X 0,Y 92.905,Z 385.023,A -85,B 0,C 180,E1 -28048.033,E2 -28048.033} C_VEL
LIN {X 0,Y 101.936,Z 380.413,A -85,B 0,C 180,E1 -28053.671,E2 -28053.671} C_VEL
LIN {X 0,Y 110.87,Z 374.689,A -85,B 0,C 180,E1 -28057.974,E2 -28057.974} C_VEL
LIN {X 0,Y 113.017,Z 373.139,A -85,B 0,C 180,E1 -28058.868,E2 -28058.868} C_VEL
LIN {X 0,Y 114.329,Z 371.528,A -85,B 0,C 180,E1 -28060.62,E2 -28060.62} C_VEL
LIN {X 0,Y 115.985,Z 367.924,A -85,B 0,C 180,E1 -28065.978,E2 -28065.978} C_VEL
LIN {X 0,Y 116.681,Z 365.915,A -85,B 0,C 180,E1 -28069.594,E2 -28069.594} C_VEL
LIN {X 0,Y 117.163,Z 364.283,A -85,B 0,C 180,E1 -28073.114,E2 -28073.114} C_VEL
LIN {X 0,Y 117.587,Z 362.979,A -85,B 0,C 180,E1 -28076.578,E2 -28076.578} C_VEL
LIN {X 0,Y 117.87,Z 362.069,A -85,B 0,C 180,E1 -28080.004,E2 -28080.004} C_VEL
LIN {X 0,Y 117.838,Z 361.78,A -85,B 0,C 180,E1 -28083.423,E2 -28083.423} C_VEL
LIN {X 0,Y 117.541,Z 362.083,A -85,B 0,C 180,E1 -28086.872,E2 -28086.872} C_VEL
LIN {X 0,Y 117.246,Z 362.773,A -85,B 0,C 180,E1 -28090.364,E2 -28090.364} C_VEL
LIN {X 0,Y 116.859,Z 364.509,A -85,B 0,C 180,E1 -28095.798,E2 -28095.798} C_VEL
LIN {X 0,Y 116.118,Z 367.215,A -85,B 0,C 180,E1 -28101.298,E2 -28101.298} C_VEL
LIN {X 0,Y 115.227,Z 369.784,A -85,B 0,C 180,E1 -28105.278,E2 -28105.278} C_VEL
LIN {X 0,Y 113.905,Z 372.958,A -85,B 0,C 180,E1 -28109.582,E2 -28109.582} C_VEL
LIN {X 0,Y 113.078,Z 374.403,A -85,B 0,C 180,E1 -28111.288,E2 -28111.288} C_VEL
LIN {X 0,Y 112.241,Z 375.459,A -85,B 0,C 180,E1 -28112.298,E2 -28112.298} C_VEL
LIN {X 0,Y 110.041,Z 377.437,A -85,B 0,C 180,E1 -28113.876,E2 -28113.876} C_VEL
LIN {X 0,Y 101.988,Z 382.716,A -85,B 0,C 180,E1 -28117.586,E2 -28117.586} C_VEL
LIN {X 0,Y 94.588,Z 386.85,A -85,B 0,C 180,E1 -28122.013,E2 -28122.013} C_VEL
LIN {X 0,Y 90.006,Z 389.054,A -85,B 0,C 180,E1 -28125.354,E2 -28125.354} C_VEL
LIN {X 0,Y 85.657,Z 390.791,A -85,B 0,C 180,E1 -28128.977,E2 -28128.977} C_VEL
LIN {X 0,Y 78.281,Z 393.087,A -85,B 0,C 180,E1 -28137.408,E2 -28137.408} C_VEL
LIN {X 0,Y 75.314,Z 393.665,A -85,B 0,C 180,E1 -28142.188,E2 -28142.188} C_VEL
LIN {X 0,Y 71.353,Z 393.61,A -85,B 0,C 180,E1 -28152.814,E2 -28152.814} C_VEL
LIN {X 0,Y 69.772,Z 392.037,A -85,B 0,C 180,E1 -28164.219,E2 -28164.219} C_VEL
LIN {X 0,Y 69.758,Z 390.632,A -85,B 0,C 180,E1 -28170,E2 -28170} C_VEL
LIN {X 0,Y 69.923,Z 387.66,A -85,B 0,C 180,E1 -28178.671,E2 -28178.671} C_VEL
LIN {X 0,Y 71.193,Z 383.6,A -85,B 0,C 180,E1 -28187.227,E2 -28187.227} C_VEL
LIN {X 0,Y 74.359,Z 377.327,A -85,B 0,C 180,E1 -28196.676,E2 -28196.676} C_VEL
LIN {X 0,Y 78.522,Z 370.484,A -85,B 0,C 180,E1 -28204.013,E2 -28204.013} C_VEL
LIN {X 0,Y 83.035,Z 362.763,A -85,B 0,C 180,E1 -28210.129,E2 -28210.129} C_VEL
LIN {X 0,Y 87.618,Z 355.015,A -85,B 0,C 180,E1 -28214.575,E2 -28214.575} C_VEL
LIN {X 0,Y 90.392,Z 346.479,A -85,B 0,C 180,E1 -28219.292,E2 -28219.292} C_VEL
LIN {X 0,Y 92.46,Z 337.927,A -85,B 0,C 180,E1 -28223.466,E2 -28223.466} C_VEL
LIN {X 0,Y 93.149,Z 333.584,A -85,B 0,C 180,E1 -28225.529,E2 -28225.529} C_VEL
LIN {X 0,Y 92.115,Z 326.552,A -85,B 0,C 180,E1 -28230.264,E2 -28230.264} C_VEL
LIN {X 0,Y 91.015,Z 322.926,A -85,B 0,C 180,E1 -28233.216,E2 -28233.216} C_VEL
LIN {X 0,Y 89.469,Z 319.244,A -85,B 0,C 180,E1 -28236.868,E2 -28236.868} C_VEL
LIN {X 0,Y 87.639,Z 315.628,A -85,B 0,C 180,E1 -28241.285,E2 -28241.285} C_VEL
LIN {X 0,Y 85.302,Z 311.155,A -85,B 0,C 180,E1 -28248.108,E2 -28248.108} C_VEL
LIN {X 0,Y 83.206,Z 307.302,A -85,B 0,C 180,E1 -28257.574,E2 -28257.574} C_VEL
LIN {X 0,Y 83.171,Z 305.937,A -85,B 0,C 180,E1 -28259.994,E2 -28259.994} C_VEL
LIN {X 0,Y 82.6,Z 306.08,A -85,B 0,C 180,E1 -28269.792,E2 -28269.792} C_VEL
LIN {X 0,Y 82.798,Z 307.346,A -85,B 0,C 180,E1 -28274.746,E2 -28274.746} C_VEL
LIN {X 0,Y 84.272,Z 310.531,A -85,B 0,C 180,E1 -28283.459,E2 -28283.459} C_VEL
LIN {X 0,Y 85.315,Z 312.034,A -85,B 0,C 180,E1 -28286.934,E2 -28286.934} C_VEL
LIN {X 0,Y 85.997,Z 313.688,A -85,B 0,C 180,E1 -28289.356,E2 -28289.356} C_VEL
LIN {X 0,Y 86.928,Z 314.91,A -85,B 0,C 180,E1 -28291.696,E2 -28291.696} C_VEL
LIN {X 0,Y 89.623,Z 320.876,A -85,B 0,C 180,E1 -28298.847,E2 -28298.847} C_VEL
LIN {X 0,Y 91.094,Z 324.596,A -85,B 0,C 180,E1 -28302.522,E2 -28302.522} C_VEL
LIN {X 0,Y 92.933,Z 330.396,A -85,B 0,C 180,E1 -28307.497,E2 -28307.497} C_VEL
LIN {X 0,Y 93.737,Z 333.996,A -85,B 0,C 180,E1 -28310.211,E2 -28310.211} C_VEL
LIN {X 0,Y 92.817,Z 341.037,A -85,B 0,C 180,E1 -28314.069,E2 -28314.069} C_VEL
